ABB RAPID module: Mod1.mod

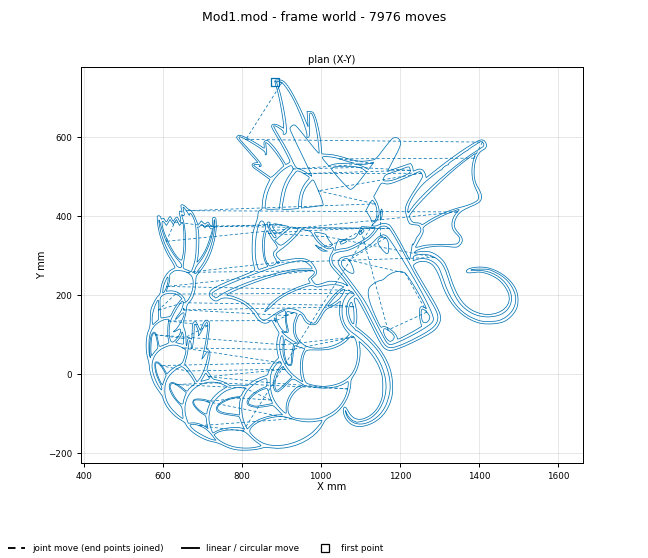
[picture p0: tool path of Mod1.mod in frame world, 7976 of 7976 moves have a stored position in this frame; points joined in program order, loops and branches not executed]
MODULE Module1
    !***********************************************************
    !
    ! Module:  Module1
    !
    ! Description:
    !   <Insert description here>
    !
    ! Author: ufabc
    !
    ! Version: 1.0
    !
    !***********************************************************


    !***********************************************************
    !
    ! Procedure main
    !
    !   This is the entry point of your program
    !
    !***********************************************************
    PROC main()
        !Add your code here
        CONST robtarget p0:=[[557.96,-192.62,509.20],[0.00299687,-0.165444,-0.986215,-0.000502744],[-1,0,0,0],[9E+09,9E+09,9E+09,9E+09,9E+09,9E+09]];	MoveJ Offs(p0,326.0,933.6, 10), v100, z1, tool0;
	MoveL Offs(p0,326.4428000000001,930.3582, 0), v100, z5, tool0;
	MoveL Offs(p0,326.7616,928.9504000000001, 0), v100, z5, tool0;
	MoveL Offs(p0,327.15,927.425, 0), v100, z5, tool0;
	MoveL Offs(p0,327.59839999999997,925.8095999999999, 0), v100, z5, tool0;
	MoveL Offs(p0,328.0972,924.1317999999999, 0), v100, z5, tool0;
	MoveL Offs(p0,328.63680000000005,922.4192, 0), v100, z5, tool0;
	MoveL Offs(p0,329.2076,920.6994000000001, 0), v100, z5, tool0;
	MoveL Offs(p0,329.8,919.0, 0), v100, z5, tool0;
	MoveL Offs(p0,331.7136,912.9074, 0), v100, z5, tool0;
	MoveL Offs(p0,333.90080000000006,904.3872000000003, 0), v100, z5, tool0;
	MoveL Offs(p0,336.25120000000004,894.0357999999999, 0), v100, z5, tool0;
	MoveL Offs(p0,338.6544,882.4496000000001, 0), v100, z5, tool0;
	MoveL Offs(p0,341.0,870.225, 0), v100, z5, tool0;
	MoveL Offs(p0,343.1776,857.9583999999999, 0), v100, z5, tool0;
	MoveL Offs(p0,345.0768,846.2461999999999, 0), v100, z5, tool0;
	MoveL Offs(p0,346.58720000000005,835.6848000000002, 0), v100, z5, tool0;
	MoveL Offs(p0,347.5984,826.8706, 0), v100, z5, tool0;
	MoveL Offs(p0,348.0,820.4, 0), v100, z5, tool0;
	MoveL Offs(p0,348.0,815.6, 0), v100, z5, tool0;
	MoveL Offs(p0,338.8,820.8, 0), v100, z5, tool0;
	MoveL Offs(p0,335.7876,822.3897999999999, 0), v100, z5, tool0;
	MoveL Offs(p0,332.98880000000014,823.6784000000001, 0), v100, z5, tool0;
	MoveL Offs(p0,330.40119999999996,824.6646000000001, 0), v100, z5, tool0;
	MoveL Offs(p0,328.0224,825.3471999999999, 0), v100, z5, tool0;
	MoveL Offs(p0,325.85,825.725, 0), v100, z5, tool0;
	MoveL Offs(p0,323.8816,825.7967999999998, 0), v100, z5, tool0;
	MoveL Offs(p0,322.11479999999995,825.5613999999999, 0), v100, z5, tool0;
	MoveL Offs(p0,320.54720000000003,825.0176000000001, 0), v100, z5, tool0;
	MoveL Offs(p0,319.1764,824.1641999999999, 0), v100, z5, tool0;
	MoveL Offs(p0,318.0,823.0, 0), v100, z5, tool0;
	MoveL Offs(p0,317.45279999999997,820.0318000000001, 0), v100, z5, tool0;
	MoveL Offs(p0,317.8976,818.4336000000001, 0), v100, z5, tool0;
	MoveL Offs(p0,318.7,816.425, 0), v100, z5, tool0;
	MoveL Offs(p0,319.8864,813.9424, 0), v100, z5, tool0;
	MoveL Offs(p0,321.4832,810.9222, 0), v100, z5, tool0;
	MoveL Offs(p0,323.51680000000005,807.3008000000001, 0), v100, z5, tool0;
	MoveL Offs(p0,326.01360000000005,803.0146000000001, 0), v100, z5, tool0;
	MoveL Offs(p0,329.0,798.0, 0), v100, z5, tool0;
	MoveL Offs(p0,333.77080000000007,789.9198000000001, 0), v100, z5, tool0;
	MoveL Offs(p0,338.63040000000007,781.4544000000002, 0), v100, z5, tool0;
	MoveL Offs(p0,343.43960000000004,772.8666000000001, 0), v100, z5, tool0;
	MoveL Offs(p0,348.05920000000003,764.4192, 0), v100, z5, tool0;
	MoveL Offs(p0,352.35,756.375, 0), v100, z5, tool0;
	MoveL Offs(p0,356.17279999999994,748.9967999999999, 0), v100, z5, tool0;
	MoveL Offs(p0,359.3884,742.5474, 0), v100, z5, tool0;
	MoveL Offs(p0,361.8576,737.2896000000001, 0), v100, z5, tool0;
	MoveL Offs(p0,363.44120000000004,733.4862, 0), v100, z5, tool0;
	MoveL Offs(p0,364.0,731.4, 0), v100, z5, tool0;
	MoveL Offs(p0,362.272,728.8313999999999, 0), v100, z5, tool0;
	MoveL Offs(p0,361.12,727.8448000000001, 0), v100, z5, tool0;
	MoveL Offs(p0,359.8,726.875, 0), v100, z5, tool0;
	MoveL Offs(p0,358.38399999999996,725.9712000000001, 0), v100, z5, tool0;
	MoveL Offs(p0,356.94399999999996,725.1826, 0), v100, z5, tool0;
	MoveL Offs(p0,355.552,724.5584000000001, 0), v100, z5, tool0;
	MoveL Offs(p0,354.28000000000003,724.1478000000001, 0), v100, z5, tool0;
	MoveL Offs(p0,353.2,724.0, 0), v100, z5, tool0;
	MoveL Offs(p0,351.7834,726.0466, 0), v100, z5, tool0;
	MoveL Offs(p0,350.82880000000006,727.5392000000002, 0), v100, z5, tool0;
	MoveL Offs(p0,349.675,729.375, 0), v100, z5, tool0;
	MoveL Offs(p0,348.34720000000004,731.5168, 0), v100, z5, tool0;
	MoveL Offs(p0,346.87059999999997,733.9273999999999, 0), v100, z5, tool0;
	MoveL Offs(p0,345.27040000000005,736.5696, 0), v100, z5, tool0;
	MoveL Offs(p0,343.5718,739.4062, 0), v100, z5, tool0;
	MoveL Offs(p0,341.8,742.4, 0), v100, z5, tool0;
	MoveL Offs(p0,339.87620000000004,745.5146000000001, 0), v100, z5, tool0;
	MoveL Offs(p0,337.73760000000004,748.8128000000003, 0), v100, z5, tool0;
	MoveL Offs(p0,335.4334,752.2262, 0), v100, z5, tool0;
	MoveL Offs(p0,333.0128,755.6864, 0), v100, z5, tool0;
	MoveL Offs(p0,330.525,759.125, 0), v100, z5, tool0;
	MoveL Offs(p0,328.0192,762.4735999999999, 0), v100, z5, tool0;
	MoveL Offs(p0,325.5446,765.6638, 0), v100, z5, tool0;
	MoveL Offs(p0,323.15040000000005,768.6272000000001, 0), v100, z5, tool0;
	MoveL Offs(p0,320.8858,771.2954000000001, 0), v100, z5, tool0;
	MoveL Offs(p0,318.8,773.6, 0), v100, z5, tool0;
	MoveL Offs(p0,315.7214,776.8180000000001, 0), v100, z5, tool0;
	MoveL Offs(p0,313.15520000000004,779.4240000000002, 0), v100, z5, tool0;
	MoveL Offs(p0,311.0258,781.466, 0), v100, z5, tool0;
	MoveL Offs(p0,309.2576,782.9920000000001, 0), v100, z5, tool0;
	MoveL Offs(p0,307.775,784.05, 0), v100, z5, tool0;
	MoveL Offs(p0,306.50239999999997,784.6879999999999, 0), v100, z5, tool0;
	MoveL Offs(p0,305.3642,784.954, 0), v100, z5, tool0;
	MoveL Offs(p0,304.2848,784.8960000000001, 0), v100, z5, tool0;
	MoveL Offs(p0,303.18860000000006,784.562, 0), v100, z5, tool0;
	MoveL Offs(p0,302.0,784.0, 0), v100, z5, tool0;
	MoveL Offs(p0,299.40079999999995,782.1351999999999, 0), v100, z5, tool0;
	MoveL Offs(p0,298.8736,781.3824000000001, 0), v100, z5, tool0;
	MoveL Offs(p0,298.5,780.5, 0), v100, z5, tool0;
	MoveL Offs(p0,298.27040000000005,779.4496, 0), v100, z5, tool0;
	MoveL Offs(p0,298.1752,778.1928, 0), v100, z5, tool0;
	MoveL Offs(p0,298.20480000000003,776.6912, 0), v100, z5, tool0;
	MoveL Offs(p0,298.3496,774.9064000000001, 0), v100, z5, tool0;
	MoveL Offs(p0,298.6,772.8, 0), v100, z5, tool0;
	MoveL Offs(p0,298.86120000000005,770.4126, 0), v100, z5, tool0;
	MoveL Offs(p0,299.0336000000001,768.5088000000003, 0), v100, z5, tool0;
	MoveL Offs(p0,299.1004,767.0562, 0), v100, z5, tool0;
	MoveL Offs(p0,299.0448,766.0224000000001, 0), v100, z5, tool0;
	MoveL Offs(p0,298.85,765.375, 0), v100, z5, tool0;
	MoveL Offs(p0,298.49920000000003,765.0815999999999, 0), v100, z5, tool0;
	MoveL Offs(p0,297.97560000000004,765.1098, 0), v100, z5, tool0;
	MoveL Offs(p0,297.2624,765.4272000000001, 0), v100, z5, tool0;
	MoveL Offs(p0,296.3428,766.0014, 0), v100, z5, tool0;
	MoveL Offs(p0,295.2,766.8, 0), v100, z5, tool0;
	MoveL Offs(p0,290.4552,770.0854000000002, 0), v100, z5, tool0;
	MoveL Offs(p0,285.0096000000001,773.6192000000003, 0), v100, z5, tool0;
	MoveL Offs(p0,279.0864,777.2778, 0), v100, z5, tool0;
	MoveL Offs(p0,272.90880000000004,780.9376000000001, 0), v100, z5, tool0;
	MoveL Offs(p0,266.7,784.475, 0), v100, z5, tool0;
	MoveL Offs(p0,260.6832,787.7663999999999, 0), v100, z5, tool0;
	MoveL Offs(p0,255.08159999999998,790.6881999999999, 0), v100, z5, tool0;
	MoveL Offs(p0,250.1184,793.1168, 0), v100, z5, tool0;
	MoveL Offs(p0,246.01680000000002,794.9286, 0), v100, z5, tool0;
	MoveL Offs(p0,243.0,796.0, 0), v100, z5, tool0;
	MoveL Offs(p0,240.78440000000006,796.5934000000001, 0), v100, z5, tool0;
	MoveL Offs(p0,238.90720000000005,797.0512000000001, 0), v100, z5, tool0;
	MoveL Offs(p0,237.3228,797.3697999999998, 0), v100, z5, tool0;
	MoveL Offs(p0,235.98559999999998,797.5456000000001, 0), v100, z5, tool0;
	MoveL Offs(p0,234.85,797.575, 0), v100, z5, tool0;
	MoveL Offs(p0,233.87039999999996,797.4544, 0), v100, z5, tool0;
	MoveL Offs(p0,233.0012,797.1802, 0), v100, z5, tool0;
	MoveL Offs(p0,232.1968,796.7488000000001, 0), v100, z5, tool0;
	MoveL Offs(p0,231.4116,796.1566, 0), v100, z5, tool0;
	MoveL Offs(p0,230.6,795.4, 0), v100, z5, tool0;
	MoveL Offs(p0,228.81260000000003,792.5002, 0), v100, z5, tool0;
	MoveL Offs(p0,229.43519999999998,790.8944, 0), v100, z5, tool0;
	MoveL Offs(p0,231.025,788.475, 0), v100, z5, tool0;
	MoveL Offs(p0,233.79680000000002,784.9456, 0), v100, z5, tool0;
	MoveL Offs(p0,237.9654,780.0098, 0), v100, z5, tool0;
	MoveL Offs(p0,243.74560000000002,773.3712000000002, 0), v100, z5, tool0;
	MoveL Offs(p0,251.35219999999998,764.7334000000001, 0), v100, z5, tool0;
	MoveL Offs(p0,261.0,753.8, 0), v100, z5, tool0;
	MoveL Offs(p0,282.8,729.0, 0), v100, z5, tool0;
	MoveL Offs(p0,276.0,728.0, 0), v100, z5, tool0;
	MoveL Offs(p0,273.33080000000007,727.4296, 0), v100, z5, tool0;
	MoveL Offs(p0,271.2064000000001,726.5808000000002, 0), v100, z5, tool0;
	MoveL Offs(p0,269.63160000000005,725.4871999999999, 0), v100, z5, tool0;
	MoveL Offs(p0,268.6112,724.1824, 0), v100, z5, tool0;
	MoveL Offs(p0,268.15,722.7, 0), v100, z5, tool0;
	MoveL Offs(p0,268.2528,721.0735999999999, 0), v100, z5, tool0;
	MoveL Offs(p0,268.9244,719.3368, 0), v100, z5, tool0;
	MoveL Offs(p0,270.1696,717.5232000000001, 0), v100, z5, tool0;
	MoveL Offs(p0,271.9932,715.6664000000001, 0), v100, z5, tool0;
	MoveL Offs(p0,274.4,713.8, 0), v100, z5, tool0;
	MoveL Offs(p0,277.2880000000001,711.8080000000002, 0), v100, z5, tool0;
	MoveL Offs(p0,279.206,710.452, 0), v100, z5, tool0;
	MoveL Offs(p0,281.37600000000003,708.9040000000001, 0), v100, z5, tool0;
	MoveL Offs(p0,283.75,707.2, 0), v100, z5, tool0;
	MoveL Offs(p0,286.28000000000003,705.376, 0), v100, z5, tool0;
	MoveL Offs(p0,288.918,703.4680000000001, 0), v100, z5, tool0;
	MoveL Offs(p0,291.61600000000004,701.5120000000001, 0), v100, z5, tool0;
	MoveL Offs(p0,294.326,699.5440000000001, 0), v100, z5, tool0;
	MoveL Offs(p0,297.0,697.6, 0), v100, z5, tool0;
	MoveL Offs(p0,313.2,685.8, 0), v100, z5, tool0;
	MoveL Offs(p0,306.6,672.4, 0), v100, z5, tool0;
	MoveL Offs(p0,304.44900000000007,667.78, 0), v100, z5, tool0;
	MoveL Offs(p0,302.4480000000001,662.8480000000002, 0), v100, z5, tool0;
	MoveL Offs(p0,300.61499999999995,657.676, 0), v100, z5, tool0;
	MoveL Offs(p0,298.96799999999996,652.336, 0), v100, z5, tool0;
	MoveL Offs(p0,297.525,646.9, 0), v100, z5, tool0;
	MoveL Offs(p0,296.304,641.44, 0), v100, z5, tool0;
	MoveL Offs(p0,295.323,636.028, 0), v100, z5, tool0;
	MoveL Offs(p0,294.6,630.7360000000001, 0), v100, z5, tool0;
	MoveL Offs(p0,294.15299999999996,625.6360000000001, 0), v100, z5, tool0;
	MoveL Offs(p0,294.0,620.8, 0), v100, z5, tool0;
	MoveL Offs(p0,293.9788,618.3684000000001, 0), v100, z5, tool0;
	MoveL Offs(p0,293.90240000000006,616.3232, 0), v100, z5, tool0;
	MoveL Offs(p0,293.7516,614.6188, 0), v100, z5, tool0;
	MoveL Offs(p0,293.5072,613.2096, 0), v100, z5, tool0;
	MoveL Offs(p0,293.15,612.05, 0), v100, z5, tool0;
	MoveL Offs(p0,292.6608,611.0944, 0), v100, z5, tool0;
	MoveL Offs(p0,292.0204,610.2972, 0), v100, z5, tool0;
	MoveL Offs(p0,291.2096,609.6128000000001, 0), v100, z5, tool0;
	MoveL Offs(p0,290.2092,608.9956, 0), v100, z5, tool0;
	MoveL Offs(p0,289.0,608.4, 0), v100, z5, tool0;
	MoveL Offs(p0,286.642,607.0985999999999, 0), v100, z5, tool0;
	MoveL Offs(p0,285.96000000000004,606.5952, 0), v100, z5, tool0;
	MoveL Offs(p0,285.35,606.075, 0), v100, z5, tool0;
	MoveL Offs(p0,284.824,605.5488, 0), v100, z5, tool0;
	MoveL Offs(p0,284.394,605.0274, 0), v100, z5, tool0;
	MoveL Offs(p0,284.072,604.5216, 0), v100, z5, tool0;
	MoveL Offs(p0,283.87,604.0422000000001, 0), v100, z5, tool0;
	MoveL Offs(p0,283.8,603.6, 0), v100, z5, tool0;
	MoveL Offs(p0,283.4896,600.7104, 0), v100, z5, tool0;
	MoveL Offs(p0,283.4,599.7, 0), v100, z5, tool0;
	MoveL Offs(p0,283.31039999999996,598.6176, 0), v100, z5, tool0;
	MoveL Offs(p0,283.2232,597.4848, 0), v100, z5, tool0;
	MoveL Offs(p0,283.1408,596.3232, 0), v100, z5, tool0;
	MoveL Offs(p0,283.0656,595.1544, 0), v100, z5, tool0;
	MoveL Offs(p0,283.0,594.0, 0), v100, z5, tool0;
	MoveL Offs(p0,282.44320000000005,590.9008000000001, 0), v100, z5, tool0;
	MoveL Offs(p0,281.9488,588.8142, 0), v100, z5, tool0;
	MoveL Offs(p0,281.3296,586.4384, 0), v100, z5, tool0;
	MoveL Offs(p0,280.6,583.825, 0), v100, z5, tool0;
	MoveL Offs(p0,279.77439999999996,581.0255999999999, 0), v100, z5, tool0;
	MoveL Offs(p0,278.8672,578.0917999999999, 0), v100, z5, tool0;
	MoveL Offs(p0,277.89279999999997,575.0752, 0), v100, z5, tool0;
	MoveL Offs(p0,276.8656,572.0274, 0), v100, z5, tool0;
	MoveL Offs(p0,275.8,569.0, 0), v100, z5, tool0;
	MoveL Offs(p0,274.1564000000001,564.3728000000001, 0), v100, z5, tool0;
	MoveL Offs(p0,272.8032000000001,560.3024000000001, 0), v100, z5, tool0;
	MoveL Offs(p0,271.7068,556.5655999999999, 0), v100, z5, tool0;
	MoveL Offs(p0,270.83360000000005,552.9392, 0), v100, z5, tool0;
	MoveL Offs(p0,270.15,549.2, 0), v100, z5, tool0;
	MoveL Offs(p0,269.62239999999997,545.1247999999999, 0), v100, z5, tool0;
	MoveL Offs(p0,269.2172,540.4904, 0), v100, z5, tool0;
	MoveL Offs(p0,268.9008,535.0735999999999, 0), v100, z5, tool0;
	MoveL Offs(p0,268.63960000000003,528.6512, 0), v100, z5, tool0;
	MoveL Offs(p0,268.4,521.0, 0), v100, z5, tool0;
	MoveL Offs(p0,268.2338000000001,512.9028000000001, 0), v100, z5, tool0;
	MoveL Offs(p0,268.22240000000005,505.56640000000016, 0), v100, z5, tool0;
	MoveL Offs(p0,268.37659999999994,498.8636, 0), v100, z5, tool0;
	MoveL Offs(p0,268.7072,492.66720000000004, 0), v100, z5, tool0;
	MoveL Offs(p0,269.225,486.85, 0), v100, z5, tool0;
	MoveL Offs(p0,269.94079999999997,481.2848, 0), v100, z5, tool0;
	MoveL Offs(p0,270.8654,475.84439999999995, 0), v100, z5, tool0;
	MoveL Offs(p0,272.00960000000003,470.4016, 0), v100, z5, tool0;
	MoveL Offs(p0,273.3842,464.8292, 0), v100, z5, tool0;
	MoveL Offs(p0,275.0,459.0, 0), v100, z5, tool0;
	MoveL Offs(p0,275.0176,456.8880000000001, 0), v100, z5, tool0;
	MoveL Offs(p0,274.30339999999995,455.85, 0), v100, z5, tool0;
	MoveL Offs(p0,272.93280000000004,454.72799999999995, 0), v100, z5, tool0;
	MoveL Offs(p0,270.775,453.45, 0), v100, z5, tool0;
	MoveL Offs(p0,267.6992,451.9440000000001, 0), v100, z5, tool0;
	MoveL Offs(p0,263.57460000000003,450.13800000000003, 0), v100, z5, tool0;
	MoveL Offs(p0,258.2704,447.96000000000004, 0), v100, z5, tool0;
	MoveL Offs(p0,251.6558,445.338, 0), v100, z5, tool0;
	MoveL Offs(p0,243.6,442.2, 0), v100, z5, tool0;
	MoveL Offs(p0,230.11380000000003,436.89400000000006, 0), v100, z5, tool0;
	MoveL Offs(p0,217.95840000000004,432.00800000000015, 0), v100, z5, tool0;
	MoveL Offs(p0,207.10859999999997,427.53000000000003, 0), v100, z5, tool0;
	MoveL Offs(p0,197.5392,423.44800000000004, 0), v100, z5, tool0;
	MoveL Offs(p0,189.225,419.75, 0), v100, z5, tool0;
	MoveL Offs(p0,182.14079999999998,416.424, 0), v100, z5, tool0;
	MoveL Offs(p0,176.2614,413.45799999999997, 0), v100, z5, tool0;
	MoveL Offs(p0,171.5616,410.84, 0), v100, z5, tool0;
	MoveL Offs(p0,168.0162,408.558, 0), v100, z5, tool0;
	MoveL Offs(p0,165.6,406.6, 0), v100, z5, tool0;
	MoveL Offs(p0,163.50000000000003,404.2816000000001, 0), v100, z5, tool0;
	MoveL Offs(p0,161.88000000000005,401.9008000000001, 0), v100, z5, tool0;
	MoveL Offs(p0,160.74,399.47919999999993, 0), v100, z5, tool0;
	MoveL Offs(p0,160.08,397.0384, 0), v100, z5, tool0;
	MoveL Offs(p0,159.9,394.6, 0), v100, z5, tool0;
	MoveL Offs(p0,160.2,392.18559999999997, 0), v100, z5, tool0;
	MoveL Offs(p0,160.98000000000002,389.81679999999994, 0), v100, z5, tool0;
	MoveL Offs(p0,162.24,387.5152, 0), v100, z5, tool0;
	MoveL Offs(p0,163.98000000000002,385.30240000000003, 0), v100, z5, tool0;
	MoveL Offs(p0,166.2,383.2, 0), v100, z5, tool0;
	MoveL Offs(p0,168.3522,381.51400000000007, 0), v100, z5, tool0;
	MoveL Offs(p0,170.38560000000007,380.17600000000004, 0), v100, z5, tool0;
	MoveL Offs(p0,172.3254,379.18600000000004, 0), v100, z5, tool0;
	MoveL Offs(p0,174.1968,378.544, 0), v100, z5, tool0;
	MoveL Offs(p0,176.025,378.25, 0), v100, z5, tool0;
	MoveL Offs(p0,177.83520000000001,378.304, 0), v100, z5, tool0;
	MoveL Offs(p0,179.65259999999998,378.706, 0), v100, z5, tool0;
	MoveL Offs(p0,181.50240000000002,379.456, 0), v100, z5, tool0;
	MoveL Offs(p0,183.40980000000002,380.554, 0), v100, z5, tool0;
	MoveL Offs(p0,185.4,382.0, 0), v100, z5, tool0;
	MoveL Offs(p0,189.10640000000004,384.06820000000005, 0), v100, z5, tool0;
	MoveL Offs(p0,193.76320000000004,385.36960000000005, 0), v100, z5, tool0;
	MoveL Offs(p0,199.21679999999998,385.9294, 0), v100, z5, tool0;
	MoveL Offs(p0,205.31360000000004,385.7728000000001, 0), v100, z5, tool0;
	MoveL Offs(p0,211.9,384.925, 0), v100, z5, tool0;
	MoveL Offs(p0,218.82240000000002,383.4112, 0), v100, z5, tool0;
	MoveL Offs(p0,225.9272,381.2566, 0), v100, z5, tool0;
	MoveL Offs(p0,233.06080000000003,378.48640000000006, 0), v100, z5, tool0;
	MoveL Offs(p0,240.06959999999998,375.12579999999997, 0), v100, z5, tool0;
	MoveL Offs(p0,246.8,371.2, 0), v100, z5, tool0;
	MoveL Offs(p0,250.31440000000003,368.80140000000006, 0), v100, z5, tool0;
	MoveL Offs(p0,253.77120000000005,366.1712000000001, 0), v100, z5, tool0;
	MoveL Offs(p0,257.1608,363.31780000000003, 0), v100, z5, tool0;
	MoveL Offs(p0,260.47360000000003,360.2496, 0), v100, z5, tool0;
	MoveL Offs(p0,263.7,356.975, 0), v100, z5, tool0;
	MoveL Offs(p0,266.8304,353.50239999999997, 0), v100, z5, tool0;
	MoveL Offs(p0,269.85519999999997,349.8402, 0), v100, z5, tool0;
	MoveL Offs(p0,272.76480000000004,345.9968, 0), v100, z5, tool0;
	MoveL Offs(p0,275.5496,341.98060000000004, 0), v100, z5, tool0;
	MoveL Offs(p0,278.2,337.8, 0), v100, z5, tool0;
	MoveL Offs(p0,281.2044,333.5006000000001, 0), v100, z5, tool0;
	MoveL Offs(p0,284.4272,329.85280000000006, 0), v100, z5, tool0;
	MoveL Offs(p0,287.82280000000003,326.8722, 0), v100, z5, tool0;
	MoveL Offs(p0,291.3456,324.5744, 0), v100, z5, tool0;
	MoveL Offs(p0,294.95,322.975, 0), v100, z5, tool0;
	MoveL Offs(p0,298.5904,322.08959999999996, 0), v100, z5, tool0;
	MoveL Offs(p0,302.2212,321.93379999999996, 0), v100, z5, tool0;
	MoveL Offs(p0,305.7968,322.5232, 0), v100, z5, tool0;
	MoveL Offs(p0,309.27160000000003,323.87340000000006, 0), v100, z5, tool0;
	MoveL Offs(p0,312.6,326.0, 0), v100, z5, tool0;
	MoveL Offs(p0,317.8,330.2, 0), v100, z5, tool0;
	MoveL Offs(p0,322.8,320.6, 0), v100, z5, tool0;
	MoveL Offs(p0,324.64480000000015,317.2416000000002, 0), v100, z5, tool0;
	MoveL Offs(p0,325.6601999999999,315.4394, 0), v100, z5, tool0;
	MoveL Offs(p0,326.71040000000005,313.6048, 0), v100, z5, tool0;
	MoveL Offs(p0,327.775,311.775, 0), v100, z5, tool0;
	MoveL Offs(p0,328.83360000000005,309.9872, 0), v100, z5, tool0;
	MoveL Offs(p0,329.8658,308.2786, 0), v100, z5, tool0;
	MoveL Offs(p0,330.85120000000006,306.68640000000005, 0), v100, z5, tool0;
	MoveL Offs(p0,331.7694,305.2478, 0), v100, z5, tool0;
	MoveL Offs(p0,332.6,304.0, 0), v100, z5, tool0;
	MoveL Offs(p0,334.74720000000013,300.7248000000001, 0), v100, z5, tool0;
	MoveL Offs(p0,335.4638,299.4172, 0), v100, z5, tool0;
	MoveL Offs(p0,335.95360000000005,298.2464, 0), v100, z5, tool0;
	MoveL Offs(p0,336.225,297.15, 0), v100, z5, tool0;
	MoveL Offs(p0,336.2864,296.0656, 0), v100, z5, tool0;
	MoveL Offs(p0,336.1462,294.9308, 0), v100, z5, tool0;
	MoveL Offs(p0,335.81280000000004,293.68320000000006, 0), v100, z5, tool0;
	MoveL Offs(p0,335.2946,292.2604, 0), v100, z5, tool0;
	MoveL Offs(p0,334.6,290.6, 0), v100, z5, tool0;
	MoveL Offs(p0,333.38820000000004,287.2198, 0), v100, z5, tool0;
	MoveL Offs(p0,332.3936000000001,283.4784000000001, 0), v100, z5, tool0;
	MoveL Offs(p0,331.6174,279.4346, 0), v100, z5, tool0;
	MoveL Offs(p0,331.0608,275.1472, 0), v100, z5, tool0;
	MoveL Offs(p0,330.725,270.675, 0), v100, z5, tool0;
	MoveL Offs(p0,330.6112,266.0768, 0), v100, z5, tool0;
	MoveL Offs(p0,330.7206,261.4114, 0), v100, z5, tool0;
	MoveL Offs(p0,331.0544,256.73760000000004, 0), v100, z5, tool0;
	MoveL Offs(p0,331.6138,252.11419999999998, 0), v100, z5, tool0;
	MoveL Offs(p0,332.4,247.6, 0), v100, z5, tool0;
	MoveL Offs(p0,335.2,234.2, 0), v100, z5, tool0;
	MoveL Offs(p0,327.6,226.6, 0), v100, z5, tool0;
	MoveL Offs(p0,325.253,224.04980000000006, 0), v100, z5, tool0;
	MoveL Offs(p0,322.72000000000014,220.83840000000004, 0), v100, z5, tool0;
	MoveL Offs(p0,320.10299999999995,217.1446, 0), v100, z5, tool0;
	MoveL Offs(p0,317.504,213.14720000000003, 0), v100, z5, tool0;
	MoveL Offs(p0,315.025,209.025, 0), v100, z5, tool0;
	MoveL Offs(p0,312.768,204.95680000000002, 0), v100, z5, tool0;
	MoveL Offs(p0,310.83500000000004,201.1214, 0), v100, z5, tool0;
	MoveL Offs(p0,309.32800000000003,197.69760000000002, 0), v100, z5, tool0;
	MoveL Offs(p0,308.349,194.8642, 0), v100, z5, tool0;
	MoveL Offs(p0,308.0,192.8, 0), v100, z5, tool0;
	MoveL Offs(p0,305.55,190.325, 0), v100, z5, tool0;
	MoveL Offs(p0,304.5872,189.8048, 0), v100, z5, tool0;
	MoveL Offs(p0,303.5116,189.3014, 0), v100, z5, tool0;
	MoveL Offs(p0,302.3424,188.8256, 0), v100, z5, tool0;
	MoveL Offs(p0,301.09880000000004,188.3882, 0), v100, z5, tool0;
	MoveL Offs(p0,299.8,188.0, 0), v100, z5, tool0;
	MoveL Offs(p0,295.9290000000001,186.8418, 0), v100, z5, tool0;
	MoveL Offs(p0,291.92,185.43040000000005, 0), v100, z5, tool0;
	MoveL Offs(p0,287.83900000000006,183.8006, 0), v100, z5, tool0;
	MoveL Offs(p0,283.752,181.98720000000003, 0), v100, z5, tool0;
	MoveL Offs(p0,279.725,180.025, 0), v100, z5, tool0;
	MoveL Offs(p0,275.82399999999996,177.9488, 0), v100, z5, tool0;
	MoveL Offs(p0,272.11499999999995,175.79339999999996, 0), v100, z5, tool0;
	MoveL Offs(p0,268.66400000000004,173.5936, 0), v100, z5, tool0;
	MoveL Offs(p0,265.53700000000003,171.38420000000002, 0), v100, z5, tool0;
	MoveL Offs(p0,262.8,169.2, 0), v100, z5, tool0;
	MoveL Offs(p0,259.1408000000001,166.16800000000003, 0), v100, z5, tool0;
	MoveL Offs(p0,257.65919999999994,165.132, 0), v100, z5, tool0;
	MoveL Offs(p0,256.27840000000003,164.38400000000001, 0), v100, z5, tool0;
	MoveL Offs(p0,254.9,163.9, 0), v100, z5, tool0;
	MoveL Offs(p0,253.42559999999997,163.656, 0), v100, z5, tool0;
	MoveL Offs(p0,251.75679999999997,163.628, 0), v100, z5, tool0;
	MoveL Offs(p0,249.79520000000002,163.792, 0), v100, z5, tool0;
	MoveL Offs(p0,247.4424,164.12400000000002, 0), v100, z5, tool0;
	MoveL Offs(p0,244.6,164.6, 0), v100, z5, tool0;
	MoveL Offs(p0,240.55040000000014,165.08000000000004, 0), v100, z5, tool0;
	MoveL Offs(p0,238.40259999999998,165.22999999999996, 0), v100, z5, tool0;
	MoveL Offs(p0,236.2032,165.32, 0), v100, z5, tool0;
	MoveL Offs(p0,233.975,165.35, 0), v100, z5, tool0;
	MoveL Offs(p0,231.74079999999998,165.32, 0), v100, z5, tool0;
	MoveL Offs(p0,229.52339999999998,165.22999999999996, 0), v100, z5, tool0;
	MoveL Offs(p0,227.34560000000002,165.08, 0), v100, z5, tool0;
	MoveL Offs(p0,225.23020000000002,164.87000000000003, 0), v100, z5, tool0;
	MoveL Offs(p0,223.2,164.6, 0), v100, z5, tool0;
	MoveL Offs(p0,220.54840000000007,164.12760000000003, 0), v100, z5, tool0;
	MoveL Offs(p0,218.30720000000005,163.79680000000005, 0), v100, z5, tool0;
	MoveL Offs(p0,216.40680000000003,163.6172, 0), v100, z5, tool0;
	MoveL Offs(p0,214.77759999999998,163.5984, 0), v100, z5, tool0;
	MoveL Offs(p0,213.35,163.75, 0), v100, z5, tool0;
	MoveL Offs(p0,212.0544,164.08160000000004, 0), v100, z5, tool0;
	MoveL Offs(p0,210.8212,164.60279999999997, 0), v100, z5, tool0;
	MoveL Offs(p0,209.5808,165.32319999999999, 0), v100, z5, tool0;
	MoveL Offs(p0,208.2636,166.25240000000002, 0), v100, z5, tool0;
	MoveL Offs(p0,206.8,167.4, 0), v100, z5, tool0;
	MoveL Offs(p0,202.48000000000005,170.23680000000004, 0), v100, z5, tool0;
	MoveL Offs(p0,199.834,171.6012, 0), v100, z5, tool0;
	MoveL Offs(p0,196.912,172.9104, 0), v100, z5, tool0;
	MoveL Offs(p0,193.75,174.15, 0), v100, z5, tool0;
	MoveL Offs(p0,190.38400000000001,175.3056, 0), v100, z5, tool0;
	MoveL Offs(p0,186.85,176.3628, 0), v100, z5, tool0;
	MoveL Offs(p0,183.18400000000003,177.30720000000002, 0), v100, z5, tool0;
	MoveL Offs(p0,179.42200000000003,178.1244, 0), v100, z5, tool0;
	MoveL Offs(p0,175.6,178.8, 0), v100, z5, tool0;
	MoveL Offs(p0,172.40960000000004,179.55200000000005, 0), v100, z5, tool0;
	MoveL Offs(p0,171.0694,180.078, 0), v100, z5, tool0;
	MoveL Offs(p0,169.85280000000003,180.73600000000002, 0), v100, z5, tool0;
	MoveL Offs(p0,168.725,181.55, 0), v100, z5, tool0;
	MoveL Offs(p0,167.6512,182.54399999999998, 0), v100, z5, tool0;
	MoveL Offs(p0,166.5966,183.74200000000002, 0), v100, z5, tool0;
	MoveL Offs(p0,165.52640000000002,185.168, 0), v100, z5, tool0;
	MoveL Offs(p0,164.4058,186.846, 0), v100, z5, tool0;
	MoveL Offs(p0,163.2,188.8, 0), v100, z5, tool0;
	MoveL Offs(p0,161.46720000000005,191.57440000000003, 0), v100, z5, tool0;
	MoveL Offs(p0,160.5828,192.9346, 0), v100, z5, tool0;
	MoveL Offs(p0,159.7056,194.24320000000003, 0), v100, z5, tool0;
	MoveL Offs(p0,158.85,195.475, 0), v100, z5, tool0;
	MoveL Offs(p0,158.03040000000001,196.6048, 0), v100, z5, tool0;
	MoveL Offs(p0,157.2612,197.60739999999998, 0), v100, z5, tool0;
	MoveL Offs(p0,156.5568,198.4576, 0), v100, z5, tool0;
	MoveL Offs(p0,155.93160000000003,199.1302, 0), v100, z5, tool0;
	MoveL Offs(p0,155.4,199.6, 0), v100, z5, tool0;
	MoveL Offs(p0,154.0176,201.89679999999998, 0), v100, z5, tool0;
	MoveL Offs(p0,153.91520000000003,203.04960000000003, 0), v100, z5, tool0;
	MoveL Offs(p0,154.0,204.5, 0), v100, z5, tool0;
	MoveL Offs(p0,154.27679999999998,206.3104, 0), v100, z5, tool0;
	MoveL Offs(p0,154.75039999999998,208.54319999999998, 0), v100, z5, tool0;
	MoveL Offs(p0,155.4256,211.26080000000002, 0), v100, z5, tool0;
	MoveL Offs(p0,156.30720000000002,214.52560000000003, 0), v100, z5, tool0;
	MoveL Offs(p0,157.4,218.4, 0), v100, z5, tool0;
	MoveL Offs(p0,158.9116,224.1442, 0), v100, z5, tool0;
	MoveL Offs(p0,160.08480000000003,229.48160000000007, 0), v100, z5, tool0;
	MoveL Offs(p0,160.91720000000004,234.38939999999997, 0), v100, z5, tool0;
	MoveL Offs(p0,161.40640000000002,238.84480000000002, 0), v100, z5, tool0;
	MoveL Offs(p0,161.55,242.825, 0), v100, z5, tool0;
	MoveL Offs(p0,161.3456,246.30720000000002, 0), v100, z5, tool0;
	MoveL Offs(p0,160.7908,249.26859999999996, 0), v100, z5, tool0;
	MoveL Offs(p0,159.8832,251.68640000000005, 0), v100, z5, tool0;
	MoveL Offs(p0,158.62040000000002,253.5378, 0), v100, z5, tool0;
	MoveL Offs(p0,157.0,254.8, 0), v100, z5, tool0;
	MoveL Offs(p0,154.5584,256.0928, 0), v100, z5, tool0;
	MoveL Offs(p0,154.05,256.35, 0), v100, z5, tool0;
	MoveL Offs(p0,153.60160000000002,256.5712, 0), v100, z5, tool0;
	MoveL Offs(p0,153.2228,256.7516, 0), v100, z5, tool0;
	MoveL Offs(p0,152.92320000000004,256.88640000000004, 0), v100, z5, tool0;
	MoveL Offs(p0,152.71240000000003,256.9708, 0), v100, z5, tool0;
	MoveL Offs(p0,152.6,257.0, 0), v100, z5, tool0;
	MoveL Offs(p0,152.95,259.975, 0), v100, z5, tool0;
	MoveL Offs(p0,153.14719999999997,261.1472, 0), v100, z5, tool0;
	MoveL Offs(p0,153.3756,262.45860000000005, 0), v100, z5, tool0;
	MoveL Offs(p0,153.6304,263.88640000000004, 0), v100, z5, tool0;
	MoveL Offs(p0,153.90680000000003,265.4078, 0), v100, z5, tool0;
	MoveL Offs(p0,154.2,267.0, 0), v100, z5, tool0;
	MoveL Offs(p0,155.00640000000004,271.37280000000004, 0), v100, z5, tool0;
	MoveL Offs(p0,155.46359999999999,274.21619999999996, 0), v100, z5, tool0;
	MoveL Offs(p0,155.9472,277.40639999999996, 0), v100, z5, tool0;
	MoveL Offs(p0,156.45,280.875, 0), v100, z5, tool0;
	MoveL Offs(p0,156.96479999999997,284.5536, 0), v100, z5, tool0;
	MoveL Offs(p0,157.4844,288.3738, 0), v100, z5, tool0;
	MoveL Offs(p0,158.0016,292.26720000000006, 0), v100, z5, tool0;
	MoveL Offs(p0,158.50920000000002,296.16540000000003, 0), v100, z5, tool0;
	MoveL Offs(p0,159.0,300.0, 0), v100, z5, tool0;
	MoveL Offs(p0,159.6474,305.7074000000001, 0), v100, z5, tool0;
	MoveL Offs(p0,160.14720000000003,310.4272000000001, 0), v100, z5, tool0;
	MoveL Offs(p0,160.49579999999997,314.2758, 0), v100, z5, tool0;
	MoveL Offs(p0,160.6896,317.36960000000005, 0), v100, z5, tool0;
	MoveL Offs(p0,160.725,319.825, 0), v100, z5, tool0;
	MoveL Offs(p0,160.59840000000003,321.7584, 0), v100, z5, tool0;
	MoveL Offs(p0,160.3062,323.2862, 0), v100, z5, tool0;
	MoveL Offs(p0,159.84480000000002,324.5248, 0), v100, z5, tool0;
	MoveL Offs(p0,159.2106,325.5906, 0), v100, z5, tool0;
	MoveL Offs(p0,158.4,326.6, 0), v100, z5, tool0;
	MoveL Offs(p0,155.0448,329.3008000000001, 0), v100, z5, tool0;
	MoveL Offs(p0,153.43919999999997,329.7842, 0), v100, z5, tool0;
	MoveL Offs(p0,151.8624,329.6784, 0), v100, z5, tool0;
	MoveL Offs(p0,150.3,328.975, 0), v100, z5, tool0;
	MoveL Offs(p0,148.7376,327.6656, 0), v100, z5, tool0;
	MoveL Offs(p0,147.1608,325.7418, 0), v100, z5, tool0;
	MoveL Offs(p0,145.5552,323.1952, 0), v100, z5, tool0;
	MoveL Offs(p0,143.90640000000002,320.0174, 0), v100, z5, tool0;
	MoveL Offs(p0,142.2,316.2, 0), v100, z5, tool0;
	MoveL Offs(p0,137.0,303.4, 0), v100, z5, tool0;
	MoveL Offs(p0,132.0,314.6, 0), v100, z5, tool0;
	MoveL Offs(p0,130.38880000000003,318.16640000000007, 0), v100, z5, tool0;
	MoveL Offs(p0,129.5682,319.7966, 0), v100, z5, tool0;
	MoveL Offs(p0,128.7584,321.2912, 0), v100, z5, tool0;
	MoveL Offs(p0,127.975,322.625, 0), v100, z5, tool0;
	MoveL Offs(p0,127.23359999999998,323.77279999999996, 0), v100, z5, tool0;
	MoveL Offs(p0,126.5498,324.7094, 0), v100, z5, tool0;
	MoveL Offs(p0,125.9392,325.4096, 0), v100, z5, tool0;
	MoveL Offs(p0,125.4174,325.8482, 0), v100, z5, tool0;
	MoveL Offs(p0,125.0,326.0, 0), v100, z5, tool0;
	MoveL Offs(p0,122.09280000000001,325.41280000000006, 0), v100, z5, tool0;
	MoveL Offs(p0,120.88520000000001,324.7562, 0), v100, z5, tool0;
	MoveL Offs(p0,119.83840000000001,323.8464, 0), v100, z5, tool0;
	MoveL Offs(p0,118.95,322.675, 0), v100, z5, tool0;
	MoveL Offs(p0,118.21759999999999,321.23359999999997, 0), v100, z5, tool0;
	MoveL Offs(p0,117.63879999999999,319.5138, 0), v100, z5, tool0;
	MoveL Offs(p0,117.2112,317.5072, 0), v100, z5, tool0;
	MoveL Offs(p0,116.9324,315.2054, 0), v100, z5, tool0;
	MoveL Offs(p0,116.8,312.6, 0), v100, z5, tool0;
	MoveL Offs(p0,116.7168,306.7532, 0), v100, z5, tool0;
	MoveL Offs(p0,116.59040000000002,301.36960000000005, 0), v100, z5, tool0;
	MoveL Offs(p0,116.42559999999999,296.5044, 0), v100, z5, tool0;
	MoveL Offs(p0,116.22720000000001,292.2128, 0), v100, z5, tool0;
	MoveL Offs(p0,116.0,288.55, 0), v100, z5, tool0;
	MoveL Offs(p0,115.7488,285.5712, 0), v100, z5, tool0;
	MoveL Offs(p0,115.47840000000001,283.33160000000004, 0), v100, z5, tool0;
	MoveL Offs(p0,115.19360000000002,281.88640000000004, 0), v100, z5, tool0;
	MoveL Offs(p0,114.8992,281.29080000000005, 0), v100, z5, tool0;
	MoveL Offs(p0,114.6,281.6, 0), v100, z5, tool0;
	MoveL Offs(p0,112.21679999999999,283.64480000000003, 0), v100, z5, tool0;
	MoveL Offs(p0,111.08960000000002,283.88160000000005, 0), v100, z5, tool0;
	MoveL Offs(p0,109.9,283.9, 0), v100, z5, tool0;
	MoveL Offs(p0,108.7104,283.7024, 0), v100, z5, tool0;
	MoveL Offs(p0,107.58319999999999,283.2912, 0), v100, z5, tool0;
	MoveL Offs(p0,106.5808,282.66880000000003, 0), v100, z5, tool0;
	MoveL Offs(p0,105.76559999999999,281.8376, 0), v100, z5, tool0;
	MoveL Offs(p0,105.2,280.8, 0), v100, z5, tool0;
	MoveL Offs(p0,104.6762,278.721, 0), v100, z5, tool0;
	MoveL Offs(p0,104.5184,277.872, 0), v100, z5, tool0;
	MoveL Offs(p0,104.375,276.975, 0), v100, z5, tool0;
	MoveL Offs(p0,104.24960000000002,276.04799999999994, 0), v100, z5, tool0;
	MoveL Offs(p0,104.14579999999998,275.10900000000004, 0), v100, z5, tool0;
	MoveL Offs(p0,104.0672,274.17600000000004, 0), v100, z5, tool0;
	MoveL Offs(p0,104.0174,273.267, 0), v100, z5, tool0;
	MoveL Offs(p0,104.0,272.4, 0), v100, z5, tool0;
	MoveL Offs(p0,103.80559999999998,269.65680000000003, 0), v100, z5, tool0;
	MoveL Offs(p0,103.66720000000001,268.7616, 0), v100, z5, tool0;
	MoveL Offs(p0,103.5,267.9, 0), v100, z5, tool0;
	MoveL Offs(p0,103.30879999999999,267.08639999999997, 0), v100, z5, tool0;
	MoveL Offs(p0,103.0984,266.3352, 0), v100, z5, tool0;
	MoveL Offs(p0,102.87360000000001,265.6608, 0), v100, z5, tool0;
	MoveL Offs(p0,102.6392,265.07759999999996, 0), v100, z5, tool0;
	MoveL Offs(p0,102.4,264.6, 0), v100, z5, tool0;
	MoveL Offs(p0,101.54880000000001,266.6544, 0), v100, z5, tool0;
	MoveL Offs(p0,101.375,268.125, 0), v100, z5, tool0;
	MoveL Offs(p0,101.2192,269.9136, 0), v100, z5, tool0;
	MoveL Offs(p0,101.0826,271.9878, 0), v100, z5, tool0;
	MoveL Offs(p0,100.96640000000001,274.3152, 0), v100, z5, tool0;
	MoveL Offs(p0,100.87180000000001,276.8634, 0), v100, z5, tool0;
	MoveL Offs(p0,100.8,279.6, 0), v100, z5, tool0;
	MoveL Offs(p0,100.76380000000002,283.04460000000006, 0), v100, z5, tool0;
	MoveL Offs(p0,100.65440000000002,286.3008000000001, 0), v100, z5, tool0;
	MoveL Offs(p0,100.4706,289.37219999999996, 0), v100, z5, tool0;
	MoveL Offs(p0,100.21120000000002,292.2624, 0), v100, z5, tool0;
	MoveL Offs(p0,99.875,294.975, 0), v100, z5, tool0;
	MoveL Offs(p0,99.46079999999999,297.5136, 0), v100, z5, tool0;
	MoveL Offs(p0,98.9674,299.8818, 0), v100, z5, tool0;
	MoveL Offs(p0,98.3936,302.08320000000003, 0), v100, z5, tool0;
	MoveL Offs(p0,97.7382,304.1214, 0), v100, z5, tool0;
	MoveL Offs(p0,97.0,306.0, 0), v100, z5, tool0;
	MoveL Offs(p0,95.81200000000001,309.19780000000003, 0), v100, z5, tool0;
	MoveL Offs(p0,94.88800000000002,312.11840000000007, 0), v100, z5, tool0;
	MoveL Offs(p0,94.228,314.83259999999996, 0), v100, z5, tool0;
	MoveL Offs(p0,93.83200000000001,317.41120000000006, 0), v100, z5, tool0;
	MoveL Offs(p0,93.7,319.925, 0), v100, z5, tool0;
	MoveL Offs(p0,93.83200000000001,322.44480000000004, 0), v100, z5, tool0;
	MoveL Offs(p0,94.228,325.0414, 0), v100, z5, tool0;
	MoveL Offs(p0,94.888,327.78560000000004, 0), v100, z5, tool0;
	MoveL Offs(p0,95.81200000000001,330.7482, 0), v100, z5, tool0;
	MoveL Offs(p0,97.0,334.0, 0), v100, z5, tool0;
	MoveL Offs(p0,98.11040000000001,337.4944000000001, 0), v100, z5, tool0;
	MoveL Offs(p0,98.6686,339.5476, 0), v100, z5, tool0;
	MoveL Offs(p0,99.2112,341.74719999999996, 0), v100, z5, tool0;
	MoveL Offs(p0,99.725,344.05, 0), v100, z5, tool0;
	MoveL Offs(p0,100.19680000000001,346.41279999999995, 0), v100, z5, tool0;
	MoveL Offs(p0,100.6134,348.7924, 0), v100, z5, tool0;
	MoveL Offs(p0,100.9616,351.1456, 0), v100, z5, tool0;
	MoveL Offs(p0,101.22820000000002,353.42920000000004, 0), v100, z5, tool0;
	MoveL Offs(p0,101.4,355.6, 0), v100, z5, tool0;
	MoveL Offs(p0,101.71020000000001,358.5570000000001, 0), v100, z5, tool0;
	MoveL Offs(p0,102.05760000000002,361.11200000000014, 0), v100, z5, tool0;
	MoveL Offs(p0,102.4674,363.33099999999996, 0), v100, z5, tool0;
	MoveL Offs(p0,102.96480000000001,365.28000000000003, 0), v100, z5, tool0;
	MoveL Offs(p0,103.575,367.025, 0), v100, z5, tool0;
	MoveL Offs(p0,104.3232,368.632, 0), v100, z5, tool0;
	MoveL Offs(p0,105.2346,370.16700000000003, 0), v100, z5, tool0;
	MoveL Offs(p0,106.3344,371.696, 0), v100, z5, tool0;
	MoveL Offs(p0,107.6478,373.285, 0), v100, z5, tool0;
	MoveL Offs(p0,109.2,375.0, 0), v100, z5, tool0;
	MoveL Offs(p0,112.06180000000002,378.39560000000006, 0), v100, z5, tool0;
	MoveL Offs(p0,114.64640000000004,382.10080000000005, 0), v100, z5, tool0;
	MoveL Offs(p0,116.9526,386.11319999999995, 0), v100, z5, tool0;
	MoveL Offs(p0,118.97920000000002,390.4304, 0), v100, z5, tool0;
	MoveL Offs(p0,120.725,395.05, 0), v100, z5, tool0;
	MoveL Offs(p0,122.18879999999999,399.9696, 0), v100, z5, tool0;
	MoveL Offs(p0,123.3694,405.18679999999995, 0), v100, z5, tool0;
	MoveL Offs(p0,124.26559999999999,410.6992, 0), v100, z5, tool0;
	MoveL Offs(p0,124.87620000000001,416.5044, 0), v100, z5, tool0;
	MoveL Offs(p0,125.2,422.6, 0), v100, z5, tool0;
	MoveL Offs(p0,125.33380000000002,426.57480000000004, 0), v100, z5, tool0;
	MoveL Offs(p0,125.50240000000004,430.01440000000014, 0), v100, z5, tool0;
	MoveL Offs(p0,125.7166,432.9716, 0), v100, z5, tool0;
	MoveL Offs(p0,125.9872,435.49920000000003, 0), v100, z5, tool0;
	MoveL Offs(p0,126.325,437.65, 0), v100, z5, tool0;
	MoveL Offs(p0,126.7408,439.4768, 0), v100, z5, tool0;
	MoveL Offs(p0,127.24539999999999,441.03239999999994, 0), v100, z5, tool0;
	MoveL Offs(p0,127.84960000000001,442.3696, 0), v100, z5, tool0;
	MoveL Offs(p0,128.5642,443.5412, 0), v100, z5, tool0;
	MoveL Offs(p0,129.4,444.6, 0), v100, z5, tool0;
	MoveL Offs(p0,132.42540000000002,448.14160000000004, 0), v100, z5, tool0;
	MoveL Offs(p0,135.57920000000004,452.10080000000005, 0), v100, z5, tool0;
	MoveL Offs(p0,138.7978,456.37919999999997, 0), v100, z5, tool0;
	MoveL Offs(p0,142.0176,460.87840000000006, 0), v100, z5, tool0;
	MoveL Offs(p0,145.175,465.5, 0), v100, z5, tool0;
	MoveL Offs(p0,148.2064,470.1456, 0), v100, z5, tool0;
	MoveL Offs(p0,151.0482,474.7168, 0), v100, z5, tool0;
	MoveL Offs(p0,153.6368,479.1152, 0), v100, z5, tool0;
	MoveL Offs(p0,155.9086,483.2424, 0), v100, z5, tool0;
	MoveL Offs(p0,157.8,487.0, 0), v100, z5, tool0;
	MoveL Offs(p0,161.40000000000003,495.21060000000006, 0), v100, z5, tool0;
	MoveL Offs(p0,164.73600000000005,504.0128000000001, 0), v100, z5, tool0;
	MoveL Offs(p0,167.772,513.2422, 0), v100, z5, tool0;
	MoveL Offs(p0,170.472,522.7344, 0), v100, z5, tool0;
	MoveL Offs(p0,172.8,532.325, 0), v100, z5, tool0;
	MoveL Offs(p0,174.72,541.8496, 0), v100, z5, tool0;
	MoveL Offs(p0,176.196,551.1438, 0), v100, z5, tool0;
	MoveL Offs(p0,177.192,560.0432000000001, 0), v100, z5, tool0;
	MoveL Offs(p0,177.672,568.3834, 0), v100, z5, tool0;
	MoveL Offs(p0,177.6,576.0, 0), v100, z5, tool0;
	MoveL Offs(p0,177.42220000000003,579.2320000000001, 0), v100, z5, tool0;
	MoveL Offs(p0,177.23360000000005,581.8880000000001, 0), v100, z5, tool0;
	MoveL Offs(p0,177.0114,584.028, 0), v100, z5, tool0;
	MoveL Offs(p0,176.7328,585.712, 0), v100, z5, tool0;
	MoveL Offs(p0,176.375,587.0, 0), v100, z5, tool0;
	MoveL Offs(p0,175.9152,587.952, 0), v100, z5, tool0;
	MoveL Offs(p0,175.3306,588.628, 0), v100, z5, tool0;
	MoveL Offs(p0,174.59840000000003,589.0880000000001, 0), v100, z5, tool0;
	MoveL Offs(p0,173.69580000000002,589.392, 0), v100, z5, tool0;
	MoveL Offs(p0,172.6,589.6, 0), v100, z5, tool0;
	MoveL Offs(p0,170.50880000000004,589.7472000000002, 0), v100, z5, tool0;
	MoveL Offs(p0,169.7542,589.5838, 0), v100, z5, tool0;
	MoveL Offs(p0,169.1664,589.1936, 0), v100, z5, tool0;
	MoveL Offs(p0,168.725,588.525, 0), v100, z5, tool0;
	MoveL Offs(p0,168.4096,587.5264, 0), v100, z5, tool0;
	MoveL Offs(p0,168.1998,586.1461999999999, 0), v100, z5, tool0;
	MoveL Offs(p0,168.0752,584.3328, 0), v100, z5, tool0;
	MoveL Offs(p0,168.01540000000003,582.0346000000001, 0), v100, z5, tool0;
	MoveL Offs(p0,168.0,579.2, 0), v100, z5, tool0;
	MoveL Offs(p0,167.9228,575.6126000000002, 0), v100, z5, tool0;
	MoveL Offs(p0,167.69440000000006,572.6528000000002, 0), v100, z5, tool0;
	MoveL Offs(p0,167.31959999999998,570.3242, 0), v100, z5, tool0;
	MoveL Offs(p0,166.8032,568.6304, 0), v100, z5, tool0;
	MoveL Offs(p0,166.15,567.575, 0), v100, z5, tool0;
	MoveL Offs(p0,165.3648,567.1616, 0), v100, z5, tool0;
	MoveL Offs(p0,164.45239999999998,567.3938, 0), v100, z5, tool0;
	MoveL Offs(p0,163.4176,568.2752, 0), v100, z5, tool0;
	MoveL Offs(p0,162.2652,569.8094, 0), v100, z5, tool0;
	MoveL Offs(p0,161.0,572.0, 0), v100, z5, tool0;
	MoveL Offs(p0,159.10400000000004,575.3456000000002, 0), v100, z5, tool0;
	MoveL Offs(p0,158.237,576.4784, 0), v100, z5, tool0;
	MoveL Offs(p0,157.40000000000003,577.2608, 0), v100, z5, tool0;
	MoveL Offs(p0,156.575,577.7, 0), v100, z5, tool0;
	MoveL Offs(p0,155.744,577.8032000000001, 0), v100, z5, tool0;
	MoveL Offs(p0,154.88899999999998,577.5776, 0), v100, z5, tool0;
	MoveL Offs(p0,153.99200000000002,577.0304000000001, 0), v100, z5, tool0;
	MoveL Offs(p0,153.03500000000003,576.1688, 0), v100, z5, tool0;
	MoveL Offs(p0,152.0,575.0, 0), v100, z5, tool0;
	MoveL Offs(p0,149.55519999999999,573.1312, 0), v100, z5, tool0;
	MoveL Offs(p0,148.95,573.15, 0), v100, z5, tool0;
	MoveL Offs(p0,148.28480000000002,573.3728, 0), v100, z5, tool0;
	MoveL Offs(p0,147.52839999999998,573.8044, 0), v100, z5, tool0;
	MoveL Offs(p0,146.64960000000002,574.4496000000001, 0), v100, z5, tool0;
	MoveL Offs(p0,145.6172,575.3131999999999, 0), v100, z5, tool0;
	MoveL Offs(p0,144.4,576.4, 0), v100, z5, tool0;
	MoveL Offs(p0,139.6,581.0, 0), v100, z5, tool0;
	MoveL Offs(p0,136.6,576.6, 0), v100, z5, tool0;
	MoveL Offs(p0,134.9638,574.4598, 0), v100, z5, tool0;
	MoveL Offs(p0,134.4336,573.8576, 0), v100, z5, tool0;
	MoveL Offs(p0,133.925,573.325, 0), v100, z5, tool0;
	MoveL Offs(p0,133.44639999999998,572.8704, 0), v100, z5, tool0;
	MoveL Offs(p0,133.00619999999998,572.5022, 0), v100, z5, tool0;
	MoveL Offs(p0,132.61280000000002,572.2288000000001, 0), v100, z5, tool0;
	MoveL Offs(p0,132.27460000000002,572.0586, 0), v100, z5, tool0;
	MoveL Offs(p0,132.0,572.0, 0), v100, z5, tool0;
	MoveL Offs(p0,130.304,574.2528, 0), v100, z5, tool0;
	MoveL Offs(p0,129.7,575.425, 0), v100, z5, tool0;
	MoveL Offs(p0,129.048,576.7952, 0), v100, z5, tool0;
	MoveL Offs(p0,128.35999999999999,578.3406, 0), v100, z5, tool0;
	MoveL Offs(p0,127.648,580.0384, 0), v100, z5, tool0;
	MoveL Offs(p0,126.924,581.8658, 0), v100, z5, tool0;
	MoveL Offs(p0,126.2,583.8, 0), v100, z5, tool0;
	MoveL Offs(p0,124.63400000000001,587.9076000000002, 0), v100, z5, tool0;
	MoveL Offs(p0,122.96000000000001,591.7968000000002, 0), v100, z5, tool0;
	MoveL Offs(p0,121.21399999999998,595.4172000000001, 0), v100, z5, tool0;
	MoveL Offs(p0,119.43200000000002,598.7184, 0), v100, z5, tool0;
	MoveL Offs(p0,117.65,601.65, 0), v100, z5, tool0;
	MoveL Offs(p0,115.904,604.1616, 0), v100, z5, tool0;
	MoveL Offs(p0,114.22999999999999,606.2028, 0), v100, z5, tool0;
	MoveL Offs(p0,112.66400000000002,607.7232, 0), v100, z5, tool0;
	MoveL Offs(p0,111.242,608.6724, 0), v100, z5, tool0;
	MoveL Offs(p0,110.0,609.0, 0), v100, z5, tool0;
	MoveL Offs(p0,107.99839999999999,609.7452000000001, 0), v100, z5, tool0;
	MoveL Offs(p0,107.1328,610.2864000000001, 0), v100, z5, tool0;
	MoveL Offs(p0,106.2,610.95, 0), v100, z5, tool0;
	MoveL Offs(p0,105.2192,611.7216000000001, 0), v100, z5, tool0;
	MoveL Offs(p0,104.2096,612.5868, 0), v100, z5, tool0;
	MoveL Offs(p0,103.1904,613.5312, 0), v100, z5, tool0;
	MoveL Offs(p0,102.1808,614.5404000000001, 0), v100, z5, tool0;
	MoveL Offs(p0,101.2,615.6, 0), v100, z5, tool0;
	MoveL Offs(p0,97.44640000000001,619.1360000000001, 0), v100, z5, tool0;
	MoveL Offs(p0,95.6146,620.3879999999999, 0), v100, z5, tool0;
	MoveL Offs(p0,93.8752,621.28, 0), v100, z5, tool0;
	MoveL Offs(p0,92.275,621.8, 0), v100, z5, tool0;
	MoveL Offs(p0,90.8608,621.9359999999999, 0), v100, z5, tool0;
	MoveL Offs(p0,89.67940000000002,621.676, 0), v100, z5, tool0;
	MoveL Offs(p0,88.7776,621.008, 0), v100, z5, tool0;
	MoveL Offs(p0,88.2022,619.9200000000001, 0), v100, z5, tool0;
	MoveL Offs(p0,88.0,618.4, 0), v100, z5, tool0;
	MoveL Offs(p0,88.20519999999999,616.1265999999999, 0), v100, z5, tool0;
	MoveL Offs(p0,88.3584,615.1392000000001, 0), v100, z5, tool0;
	MoveL Offs(p0,88.55,614.075, 0), v100, z5, tool0;
	MoveL Offs(p0,88.77759999999999,612.9567999999999, 0), v100, z5, tool0;
	MoveL Offs(p0,89.0388,611.8074, 0), v100, z5, tool0;
	MoveL Offs(p0,89.33120000000001,610.6496000000001, 0), v100, z5, tool0;
	MoveL Offs(p0,89.65240000000001,609.5062, 0), v100, z5, tool0;
	MoveL Offs(p0,90.0,608.4, 0), v100, z5, tool0;
	MoveL Offs(p0,90.74080000000002,605.5232000000002, 0), v100, z5, tool0;
	MoveL Offs(p0,90.9432,604.5138, 0), v100, z5, tool0;
	MoveL Offs(p0,91.03040000000001,603.7696000000001, 0), v100, z5, tool0;
	MoveL Offs(p0,91.0,603.275, 0), v100, z5, tool0;
	MoveL Offs(p0,90.8496,603.0143999999999, 0), v100, z5, tool0;
	MoveL Offs(p0,90.5768,602.9721999999999, 0), v100, z5, tool0;
	MoveL Offs(p0,90.17920000000001,603.1328000000001, 0), v100, z5, tool0;
	MoveL Offs(p0,89.6544,603.4806000000001, 0), v100, z5, tool0;
	MoveL Offs(p0,89.0,604.0, 0), v100, z5, tool0;
	MoveL Offs(p0,86.32160000000002,605.6304000000002, 0), v100, z5, tool0;
	MoveL Offs(p0,85.3244,605.7135999999999, 0), v100, z5, tool0;
	MoveL Offs(p0,84.5648,605.3312000000001, 0), v100, z5, tool0;
	MoveL Offs(p0,84.05,604.5, 0), v100, z5, tool0;
	MoveL Offs(p0,83.7872,603.2367999999999, 0), v100, z5, tool0;
	MoveL Offs(p0,83.7836,601.5584, 0), v100, z5, tool0;
	MoveL Offs(p0,84.04640000000002,599.4816000000001, 0), v100, z5, tool0;
	MoveL Offs(p0,84.58279999999999,597.0232000000001, 0), v100, z5, tool0;
	MoveL Offs(p0,85.4,594.2, 0), v100, z5, tool0;
	MoveL Offs(p0,86.35520000000002,590.9248000000001, 0), v100, z5, tool0;
	MoveL Offs(p0,86.7338,589.3022, 0), v100, z5, tool0;
	MoveL Offs(p0,87.0416,587.7264000000001, 0), v100, z5, tool0;
	MoveL Offs(p0,87.275,586.225, 0), v100, z5, tool0;
	MoveL Offs(p0,87.43039999999999,584.8255999999999, 0), v100, z5, tool0;
	MoveL Offs(p0,87.5042,583.5558, 0), v100, z5, tool0;
	MoveL Offs(p0,87.49280000000002,582.4432, 0), v100, z5, tool0;
	MoveL Offs(p0,87.3926,581.5154, 0), v100, z5, tool0;
	MoveL Offs(p0,87.2,580.8, 0), v100, z5, tool0;
	MoveL Offs(p0,86.12899999999999,578.7983999999999, 0), v100, z5, tool0;
	MoveL Offs(p0,85.808,578.6208000000001, 0), v100, z5, tool0;
	MoveL Offs(p0,85.475,578.7, 0), v100, z5, tool0;
	MoveL Offs(p0,85.112,579.0432, 0), v100, z5, tool0;
	MoveL Offs(p0,84.701,579.6576, 0), v100, z5, tool0;
	MoveL Offs(p0,84.224,580.5504000000001, 0), v100, z5, tool0;
	MoveL Offs(p0,83.663,581.7288000000001, 0), v100, z5, tool0;
	MoveL Offs(p0,83.0,583.2, 0), v100, z5, tool0;
	MoveL Offs(p0,81.90400000000001,585.6486000000001, 0), v100, z5, tool0;
	MoveL Offs(p0,80.88000000000002,587.5968, 0), v100, z5, tool0;
	MoveL Offs(p0,79.904,589.0482, 0), v100, z5, tool0;
	MoveL Offs(p0,78.952,590.0064, 0), v100, z5, tool0;
	MoveL Offs(p0,78.0,590.475, 0), v100, z5, tool0;
	MoveL Offs(p0,77.024,590.4576, 0), v100, z5, tool0;
	MoveL Offs(p0,76.0,589.9577999999999, 0), v100, z5, tool0;
	MoveL Offs(p0,74.90400000000001,588.9792, 0), v100, z5, tool0;
	MoveL Offs(p0,73.712,587.5254, 0), v100, z5, tool0;
	MoveL Offs(p0,72.4,585.6, 0), v100, z5, tool0;
	MoveL Offs(p0,68.4,579.4, 0), v100, z5, tool0;
	MoveL Offs(p0,65.2,585.6, 0), v100, z5, tool0;
	MoveL Offs(p0,64.08640000000003,587.648, 0), v100, z5, tool0;
	MoveL Offs(p0,63.52059999999999,588.5699999999999, 0), v100, z5, tool0;
	MoveL Offs(p0,62.96320000000001,589.4080000000001, 0), v100, z5, tool0;
	MoveL Offs(p0,62.425,590.15, 0), v100, z5, tool0;
	MoveL Offs(p0,61.9168,590.784, 0), v100, z5, tool0;
	MoveL Offs(p0,61.449400000000004,591.298, 0), v100, z5, tool0;
	MoveL Offs(p0,61.0336,591.6800000000001, 0), v100, z5, tool0;
	MoveL Offs(p0,60.6802,591.918, 0), v100, z5, tool0;
	MoveL Offs(p0,60.4,592.0, 0), v100, z5, tool0;
	MoveL Offs(p0,58.175,589.8, 0), v100, z5, tool0;
	MoveL Offs(p0,57.606399999999994,588.9327999999999, 0), v100, z5, tool0;
	MoveL Offs(p0,57.01619999999999,587.9624, 0), v100, z5, tool0;
	MoveL Offs(p0,56.412800000000004,586.9056, 0), v100, z5, tool0;
	MoveL Offs(p0,55.80460000000001,585.7792000000001, 0), v100, z5, tool0;
	MoveL Offs(p0,55.2,584.6, 0), v100, z5, tool0;
	MoveL Offs(p0,53.47840000000002,581.1904000000002, 0), v100, z5, tool0;
	MoveL Offs(p0,52.8096,580.0495999999999, 0), v100, z5, tool0;
	MoveL Offs(p0,52.2272,579.2592000000002, 0), v100, z5, tool0;
	MoveL Offs(p0,51.7,578.8, 0), v100, z5, tool0;
	MoveL Offs(p0,51.1968,578.6528000000001, 0), v100, z5, tool0;
	MoveL Offs(p0,50.686400000000006,578.7983999999999, 0), v100, z5, tool0;
	MoveL Offs(p0,50.137600000000006,579.2176000000001, 0), v100, z5, tool0;
	MoveL Offs(p0,49.5192,579.8912, 0), v100, z5, tool0;
	MoveL Offs(p0,48.8,580.8, 0), v100, z5, tool0;
	MoveL Offs(p0,47.113600000000005,583.4304, 0), v100, z5, tool0;
	MoveL Offs(p0,46.725,584.1, 0), v100, z5, tool0;
	MoveL Offs(p0,46.3664,584.7456, 0), v100, z5, tool0;
	MoveL Offs(p0,46.0462,585.3527999999999, 0), v100, z5, tool0;
	MoveL Offs(p0,45.772800000000004,585.9072, 0), v100, z5, tool0;
	MoveL Offs(p0,45.55460000000001,586.3944, 0), v100, z5, tool0;
	MoveL Offs(p0,45.4,586.8, 0), v100, z5, tool0;
	MoveL Offs(p0,43.2776,587.5826, 0), v100, z5, tool0;
	MoveL Offs(p0,42.78240000000001,587.2864000000002, 0), v100, z5, tool0;
	MoveL Offs(p0,42.2248,586.8918000000001, 0), v100, z5, tool0;
	MoveL Offs(p0,41.6,586.4, 0), v100, z5, tool0;
	MoveL Offs(p0,39.216,585.0975999999999, 0), v100, z5, tool0;
	MoveL Offs(p0,38.8,585.225, 0), v100, z5, tool0;
	MoveL Offs(p0,38.432,585.5504, 0), v100, z5, tool0;
	MoveL Offs(p0,38.1,586.0822000000001, 0), v100, z5, tool0;
	MoveL Offs(p0,37.79200000000001,586.8288, 0), v100, z5, tool0;
	MoveL Offs(p0,37.496,587.7986, 0), v100, z5, tool0;
	MoveL Offs(p0,37.2,589.0, 0), v100, z5, tool0;
	MoveL Offs(p0,36.2046,591.5793999999999, 0), v100, z5, tool0;
	MoveL Offs(p0,35.74720000000001,592.2288000000001, 0), v100, z5, tool0;
	MoveL Offs(p0,35.225,592.775, 0), v100, z5, tool0;
	MoveL Offs(p0,34.6368,593.2192, 0), v100, z5, tool0;
	MoveL Offs(p0,33.9814,593.5626, 0), v100, z5, tool0;
	MoveL Offs(p0,33.257600000000004,593.8064, 0), v100, z5, tool0;
	MoveL Offs(p0,32.4642,593.9518, 0), v100, z5, tool0;
	MoveL Offs(p0,31.6,594.0, 0), v100, z5, tool0;
	MoveL Offs(p0,28.961199999999998,593.4707999999998, 0), v100, z5, tool0;
	MoveL Offs(p0,28.4704,592.8416, 0), v100, z5, tool0;
	MoveL Offs(p0,28.15,591.85, 0), v100, z5, tool0;
	MoveL Offs(p0,27.985599999999998,590.4143999999999, 0), v100, z5, tool0;
	MoveL Offs(p0,27.962799999999998,588.4531999999999, 0), v100, z5, tool0;
	MoveL Offs(p0,28.067200000000003,585.8848, 0), v100, z5, tool0;
	MoveL Offs(p0,28.284400000000005,582.6276, 0), v100, z5, tool0;
	MoveL Offs(p0,28.6,578.6, 0), v100, z5, tool0;
	MoveL Offs(p0,29.609400000000004,569.6076000000002, 0), v100, z5, tool0;
	MoveL Offs(p0,31.179200000000016,560.3248000000002, 0), v100, z5, tool0;
	MoveL Offs(p0,33.281800000000004,550.8331999999999, 0), v100, z5, tool0;
	MoveL Offs(p0,35.8896,541.2144000000001, 0), v100, z5, tool0;
	MoveL Offs(p0,38.975,531.55, 0), v100, z5, tool0;
	MoveL Offs(p0,42.510400000000004,521.9216, 0), v100, z5, tool0;
	MoveL Offs(p0,46.4682,512.4108, 0), v100, z5, tool0;
	MoveL Offs(p0,50.820800000000006,503.0992, 0), v100, z5, tool0;
	MoveL Offs(p0,55.540600000000005,494.0684, 0), v100, z5, tool0;
	MoveL Offs(p0,60.6,485.4, 0), v100, z5, tool0;
	MoveL Offs(p0,64.59220000000002,478.9264, 0), v100, z5, tool0;
	MoveL Offs(p0,67.72160000000002,473.7872000000002, 0), v100, z5, tool0;
	MoveL Offs(p0,70.0374,469.80480000000006, 0), v100, z5, tool0;
	MoveL Offs(p0,71.5888,466.8016000000001, 0), v100, z5, tool0;
	MoveL Offs(p0,72.425,464.6, 0), v100, z5, tool0;
	MoveL Offs(p0,72.5952,463.0224, 0), v100, z5, tool0;
	MoveL Offs(p0,72.1486,461.8912, 0), v100, z5, tool0;
	MoveL Offs(p0,71.1344,461.02880000000005, 0), v100, z5, tool0;
	MoveL Offs(p0,69.6018,460.2576, 0), v100, z5, tool0;
	MoveL Offs(p0,67.6,459.4, 0), v100, z5, tool0;
	MoveL Offs(p0,63.1792,457.0418000000001, 0), v100, z5, tool0;
	MoveL Offs(p0,58.94560000000001,453.85440000000017, 0), v100, z5, tool0;
	MoveL Offs(p0,54.9424,449.90860000000004, 0), v100, z5, tool0;
	MoveL Offs(p0,51.212800000000016,445.27520000000004, 0), v100, z5, tool0;
	MoveL Offs(p0,47.8,440.025, 0), v100, z5, tool0;
	MoveL Offs(p0,44.7472,434.22880000000004, 0), v100, z5, tool0;
	MoveL Offs(p0,42.09759999999999,427.95739999999995, 0), v100, z5, tool0;
	MoveL Offs(p0,39.894400000000005,421.2816000000001, 0), v100, z5, tool0;
	MoveL Offs(p0,38.1808,414.2722, 0), v100, z5, tool0;
	MoveL Offs(p0,37.0,407.0, 0), v100, z5, tool0;
	MoveL Offs(p0,36.6266,404.45180000000005, 0), v100, z5, tool0;
	MoveL Offs(p0,36.22080000000001,402.19040000000007, 0), v100, z5, tool0;
	MoveL Offs(p0,35.77420000000001,400.19059999999996, 0), v100, z5, tool0;
	MoveL Offs(p0,35.2784,398.42719999999997, 0), v100, z5, tool0;
	MoveL Offs(p0,34.725,396.875, 0), v100, z5, tool0;
	MoveL Offs(p0,34.105599999999995,395.5088, 0), v100, z5, tool0;
	MoveL Offs(p0,33.4118,394.3034, 0), v100, z5, tool0;
	MoveL Offs(p0,32.635200000000005,393.2336, 0), v100, z5, tool0;
	MoveL Offs(p0,31.767400000000002,392.2742, 0), v100, z5, tool0;
	MoveL Offs(p0,30.8,391.4, 0), v100, z5, tool0;
	MoveL Offs(p0,27.811999999999994,388.04479999999995, 0), v100, z5, tool0;
	MoveL Offs(p0,26.592000000000002,386.3376, 0), v100, z5, tool0;
	MoveL Offs(p0,25.3,384.4, 0), v100, z5, tool0;
	MoveL Offs(p0,23.96,382.2704, 0), v100, z5, tool0;
	MoveL Offs(p0,22.595999999999997,379.9871999999999, 0), v100, z5, tool0;
	MoveL Offs(p0,21.232000000000003,377.5888, 0), v100, z5, tool0;
	MoveL Offs(p0,19.892000000000003,375.1136, 0), v100, z5, tool0;
	MoveL Offs(p0,18.6,372.6, 0), v100, z5, tool0;
	MoveL Offs(p0,16.6372,368.52880000000005, 0), v100, z5, tool0;
	MoveL Offs(p0,15.041600000000006,365.0624000000001, 0), v100, z5, tool0;
	MoveL Offs(p0,13.7724,362.00159999999994, 0), v100, z5, tool0;
	MoveL Offs(p0,12.788800000000002,359.14720000000005, 0), v100, z5, tool0;
	MoveL Offs(p0,12.05,356.3, 0), v100, z5, tool0;
	MoveL Offs(p0,11.5152,353.2608, 0), v100, z5, tool0;
	MoveL Offs(p0,11.143600000000001,349.8304, 0), v100, z5, tool0;
	MoveL Offs(p0,10.894400000000001,345.80960000000005, 0), v100, z5, tool0;
	MoveL Offs(p0,10.7268,340.99920000000003, 0), v100, z5, tool0;
	MoveL Offs(p0,10.6,335.2, 0), v100, z5, tool0;
	MoveL Offs(p0,10.514200000000002,330.09720000000004, 0), v100, z5, tool0;
	MoveL Offs(p0,10.369600000000002,325.6496000000001, 0), v100, z5, tool0;
	MoveL Offs(p0,10.155399999999998,321.7684, 0), v100, z5, tool0;
	MoveL Offs(p0,9.860800000000001,318.3648, 0), v100, z5, tool0;
	MoveL Offs(p0,9.475,315.35, 0), v100, z5, tool0;
	MoveL Offs(p0,8.9872,312.6352, 0), v100, z5, tool0;
	MoveL Offs(p0,8.3866,310.1316, 0), v100, z5, tool0;
	MoveL Offs(p0,7.662400000000001,307.7504, 0), v100, z5, tool0;
	MoveL Offs(p0,6.8038,305.4028, 0), v100, z5, tool0;
	MoveL Offs(p0,5.8,303.0, 0), v100, z5, tool0;
	MoveL Offs(p0,3.935,297.94700000000006, 0), v100, z5, tool0;
	MoveL Offs(p0,2.4240000000000004,291.92800000000005, 0), v100, z5, tool0;
	MoveL Offs(p0,1.2729999999999992,285.15299999999996, 0), v100, z5, tool0;
	MoveL Offs(p0,0.4879999999999998,277.832, 0), v100, z5, tool0;
	MoveL Offs(p0,0.075,270.175, 0), v100, z5, tool0;
	MoveL Offs(p0,0.040000000000000216,262.392, 0), v100, z5, tool0;
	MoveL Offs(p0,0.38900000000000023,254.69299999999998, 0), v100, z5, tool0;
	MoveL Offs(p0,1.1280000000000003,247.288, 0), v100, z5, tool0;
	MoveL Offs(p0,2.263000000000001,240.387, 0), v100, z5, tool0;
	MoveL Offs(p0,3.8,234.2, 0), v100, z5, tool0;
	MoveL Offs(p0,4.500800000000001,231.844, 0), v100, z5, tool0;
	MoveL Offs(p0,5.158400000000001,229.36800000000008, 0), v100, z5, tool0;
	MoveL Offs(p0,5.765600000000001,226.82, 0), v100, z5, tool0;
	MoveL Offs(p0,6.315200000000002,224.248, 0), v100, z5, tool0;
	MoveL Offs(p0,6.8,221.7, 0), v100, z5, tool0;
	MoveL Offs(p0,7.212800000000001,219.224, 0), v100, z5, tool0;
	MoveL Offs(p0,7.5464,216.868, 0), v100, z5, tool0;
	MoveL Offs(p0,7.7936000000000005,214.68, 0), v100, z5, tool0;
	MoveL Offs(p0,7.9472000000000005,212.708, 0), v100, z5, tool0;
	MoveL Offs(p0,8.0,211.0, 0), v100, z5, tool0;
	MoveL Offs(p0,8.2306,207.497, 0), v100, z5, tool0;
	MoveL Offs(p0,8.884800000000002,203.23200000000003, 0), v100, z5, tool0;
	MoveL Offs(p0,9.906200000000002,198.391, 0), v100, z5, tool0;
	MoveL Offs(p0,11.238400000000002,193.16000000000003, 0), v100, z5, tool0;
	MoveL Offs(p0,12.825,187.725, 0), v100, z5, tool0;
	MoveL Offs(p0,14.609600000000004,182.272, 0), v100, z5, tool0;
	MoveL Offs(p0,16.535800000000002,176.987, 0), v100, z5, tool0;
	MoveL Offs(p0,18.547200000000004,172.05599999999998, 0), v100, z5, tool0;
	MoveL Offs(p0,20.587400000000002,167.66500000000002, 0), v100, z5, tool0;
	MoveL Offs(p0,22.6,164.0, 0), v100, z5, tool0;
	MoveL Offs(p0,24.26880000000001,161.31200000000007, 0), v100, z5, tool0;
	MoveL Offs(p0,25.3252,159.71599999999998, 0), v100, z5, tool0;
	MoveL Offs(p0,26.494400000000002,158.00000000000003, 0), v100, z5, tool0;
	MoveL Offs(p0,27.75,156.2, 0), v100, z5, tool0;
	MoveL Offs(p0,29.0656,154.352, 0), v100, z5, tool0;
	MoveL Offs(p0,30.414799999999996,152.49200000000002, 0), v100, z5, tool0;
	MoveL Offs(p0,31.771200000000004,150.656, 0), v100, z5, tool0;
	MoveL Offs(p0,33.1084,148.88000000000002, 0), v100, z5, tool0;
	MoveL Offs(p0,34.4,147.2, 0), v100, z5, tool0;
	MoveL Offs(p0,36.80320000000001,143.94720000000004, 0), v100, z5, tool0;
	MoveL Offs(p0,37.8938,142.3508, 0), v100, z5, tool0;
	MoveL Offs(p0,38.889599999999994,140.8096, 0), v100, z5, tool0;
	MoveL Offs(p0,39.775,139.35, 0), v100, z5, tool0;
	MoveL Offs(p0,40.53439999999999,137.9984, 0), v100, z5, tool0;
	MoveL Offs(p0,41.15220000000001,136.78119999999998, 0), v100, z5, tool0;
	MoveL Offs(p0,41.61280000000001,135.72480000000002, 0), v100, z5, tool0;
	MoveL Offs(p0,41.900600000000004,134.8556, 0), v100, z5, tool0;
	MoveL Offs(p0,42.0,134.2, 0), v100, z5, tool0;
	MoveL Offs(p0,42.65339999999999,131.3164, 0), v100, z5, tool0;
	MoveL Offs(p0,43.13280000000001,129.87680000000003, 0), v100, z5, tool0;
	MoveL Offs(p0,43.725,128.25, 0), v100, z5, tool0;
	MoveL Offs(p0,44.419200000000004,126.4672, 0), v100, z5, tool0;
	MoveL Offs(p0,45.2046,124.5596, 0), v100, z5, tool0;
	MoveL Offs(p0,46.07040000000001,122.55840000000003, 0), v100, z5, tool0;
	MoveL Offs(p0,47.00580000000001,120.49480000000001, 0), v100, z5, tool0;
	MoveL Offs(p0,48.0,118.4, 0), v100, z5, tool0;
	MoveL Offs(p0,50.463800000000006,113.75280000000001, 0), v100, z5, tool0;
	MoveL Offs(p0,53.47840000000001,108.99040000000005, 0), v100, z5, tool0;
	MoveL Offs(p0,56.95859999999999,104.20159999999998, 0), v100, z5, tool0;
	MoveL Offs(p0,60.8192,99.4752, 0), v100, z5, tool0;
	MoveL Offs(p0,64.975,94.9, 0), v100, z5, tool0;
	MoveL Offs(p0,69.3408,90.56479999999999, 0), v100, z5, tool0;
	MoveL Offs(p0,73.8314,86.55839999999999, 0), v100, z5, tool0;
	MoveL Offs(p0,78.36160000000001,82.96960000000001, 0), v100, z5, tool0;
	MoveL Offs(p0,82.84620000000001,79.8872, 0), v100, z5, tool0;
	MoveL Offs(p0,87.2,77.4, 0), v100, z5, tool0;
	MoveL Offs(p0,90.50560000000003,75.55200000000002, 0), v100, z5, tool0;
	MoveL Offs(p0,92.08340000000001,74.52899999999998, 0), v100, z5, tool0;
	MoveL Offs(p0,93.58080000000001,73.46400000000001, 0), v100, z5, tool0;
	MoveL Offs(p0,94.975,72.375, 0), v100, z5, tool0;
	MoveL Offs(p0,96.24319999999999,71.28, 0), v100, z5, tool0;
	MoveL Offs(p0,97.3626,70.197, 0), v100, z5, tool0;
	MoveL Offs(p0,98.3104,69.144, 0), v100, z5, tool0;
	MoveL Offs(p0,99.0638,68.139, 0), v100, z5, tool0;
	MoveL Offs(p0,99.6,67.2, 0), v100, z5, tool0;
	MoveL Offs(p0,102.99340000000002,61.2626, 0), v100, z5, tool0;
	MoveL Offs(p0,107.76320000000003,55.29280000000002, 0), v100, z5, tool0;
	MoveL Offs(p0,113.71379999999999,49.414199999999994, 0), v100, z5, tool0;
	MoveL Offs(p0,120.6496,43.7504, 0), v100, z5, tool0;
	MoveL Offs(p0,128.375,38.425, 0), v100, z5, tool0;
	MoveL Offs(p0,136.6944,33.5616, 0), v100, z5, tool0;
	MoveL Offs(p0,145.4122,29.283799999999996, 0), v100, z5, tool0;
	MoveL Offs(p0,154.33280000000002,25.7152, 0), v100, z5, tool0;
	MoveL Offs(p0,163.2606,22.979400000000002, 0), v100, z5, tool0;
	MoveL Offs(p0,172.0,21.2, 0), v100, z5, tool0;
	MoveL Offs(p0,175.58240000000004,20.384000000000007, 0), v100, z5, tool0;
	MoveL Offs(p0,177.7366,19.750999999999998, 0), v100, z5, tool0;
	MoveL Offs(p0,180.0672,18.992, 0), v100, z5, tool0;
	MoveL Offs(p0,182.525,18.125, 0), v100, z5, tool0;
	MoveL Offs(p0,185.06080000000003,17.168, 0), v100, z5, tool0;
	MoveL Offs(p0,187.62539999999998,16.139, 0), v100, z5, tool0;
	MoveL Offs(p0,190.1696,15.056000000000001, 0), v100, z5, tool0;
	MoveL Offs(p0,192.6442,13.937000000000001, 0), v100, z5, tool0;
	MoveL Offs(p0,195.0,12.8, 0), v100, z5, tool0;
	MoveL Offs(p0,201.3864,9.8016, 0), v100, z5, tool0;
	MoveL Offs(p0,207.42720000000003,7.268800000000003, 0), v100, z5, tool0;
	MoveL Offs(p0,213.24479999999994,5.1751999999999985, 0), v100, z5, tool0;
	MoveL Offs(p0,218.9616,3.4943999999999997, 0), v100, z5, tool0;
	MoveL Offs(p0,224.7,2.2, 0), v100, z5, tool0;
	MoveL Offs(p0,230.5824,1.2655999999999994, 0), v100, z5, tool0;
	MoveL Offs(p0,236.7312,0.6647999999999997, 0), v100, z5, tool0;
	MoveL Offs(p0,243.2688,0.3711999999999999, 0), v100, z5, tool0;
	MoveL Offs(p0,250.3176,0.35840000000000005, 0), v100, z5, tool0;
	MoveL Offs(p0,258.0,0.6, 0), v100, z5, tool0;
	MoveL Offs(p0,262.10940000000005,0.8150000000000002, 0), v100, z5, tool0;
	MoveL Offs(p0,266.13120000000004,1.0960000000000003, 0), v100, z5, tool0;
	MoveL Offs(p0,270.02579999999995,1.437, 0), v100, z5, tool0;
	MoveL Offs(p0,273.75360000000006,1.832, 0), v100, z5, tool0;
	MoveL Offs(p0,277.275,2.275, 0), v100, z5, tool0;
	MoveL Offs(p0,280.55039999999997,2.7600000000000002, 0), v100, z5, tool0;
	MoveL Offs(p0,283.5402,3.281, 0), v100, z5, tool0;
	MoveL Offs(p0,286.20480000000003,3.8320000000000007, 0), v100, z5, tool0;
	MoveL Offs(p0,288.5046,4.407, 0), v100, z5, tool0;
	MoveL Offs(p0,290.4,5.0, 0), v100, z5, tool0;
	MoveL Offs(p0,292.74260000000004,5.8112, 0), v100, z5, tool0;
	MoveL Offs(p0,294.90880000000004,6.449600000000001, 0), v100, z5, tool0;
	MoveL Offs(p0,296.98619999999994,6.9224000000000006, 0), v100, z5, tool0;
	MoveL Offs(p0,299.0624,7.236800000000001, 0), v100, z5, tool0;
	MoveL Offs(p0,301.225,7.4, 0), v100, z5, tool0;
	MoveL Offs(p0,303.5616,7.419200000000001, 0), v100, z5, tool0;
	MoveL Offs(p0,306.1598,7.301599999999999, 0), v100, z5, tool0;
	MoveL Offs(p0,309.10720000000003,7.054400000000001, 0), v100, z5, tool0;
	MoveL Offs(p0,312.4914,6.6848, 0), v100, z5, tool0;
	MoveL Offs(p0,316.4,6.2, 0), v100, z5, tool0;
	MoveL Offs(p0,332.30060000000003,5.133800000000001, 0), v100, z5, tool0;
	MoveL Offs(p0,348.3728000000001,6.046400000000001, 0), v100, z5, tool0;
	MoveL Offs(p0,364.3322,8.8046, 0), v100, z5, tool0;
	MoveL Offs(p0,379.8944,13.275200000000002, 0), v100, z5, tool0;
	MoveL Offs(p0,394.775,19.325, 0), v100, z5, tool0;
	MoveL Offs(p0,408.68960000000004,26.82080000000001, 0), v100, z5, tool0;
	MoveL Offs(p0,421.35380000000004,35.62940000000001, 0), v100, z5, tool0;
	MoveL Offs(p0,432.4832,45.61760000000001, 0), v100, z5, tool0;
	MoveL Offs(p0,441.7934,56.65220000000001, 0), v100, z5, tool0;
	MoveL Offs(p0,449.0,68.6, 0), v100, z5, tool0;
	MoveL Offs(p0,450.2706,71.10640000000001, 0), v100, z5, tool0;
	MoveL Offs(p0,451.48480000000006,73.26720000000002, 0), v100, z5, tool0;
	MoveL Offs(p0,452.70619999999997,75.14479999999999, 0), v100, z5, tool0;
	MoveL Offs(p0,453.99840000000006,76.80160000000001, 0), v100, z5, tool0;
	MoveL Offs(p0,455.425,78.3, 0), v100, z5, tool0;
	MoveL Offs(p0,457.0496,79.7024, 0), v100, z5, tool0;
	MoveL Offs(p0,458.93580000000003,81.0712, 0), v100, z5, tool0;
	MoveL Offs(p0,461.1472,82.46880000000002, 0), v100, z5, tool0;
	MoveL Offs(p0,463.7474,83.9576, 0), v100, z5, tool0;
	MoveL Offs(p0,466.8,85.6, 0), v100, z5, tool0;
	MoveL Offs(p0,475.22660000000013,90.73440000000002, 0), v100, z5, tool0;
	MoveL Offs(p0,483.1648,97.03520000000002, 0), v100, z5, tool0;
	MoveL Offs(p0,490.5221999999999,104.34880000000001, 0), v100, z5, tool0;
	MoveL Offs(p0,497.20640000000003,112.5216, 0), v100, z5, tool0;
	MoveL Offs(p0,503.125,121.4, 0), v100, z5, tool0;
	MoveL Offs(p0,508.18559999999997,130.8304, 0), v100, z5, tool0;
	MoveL Offs(p0,512.2958000000001,140.6592, 0), v100, z5, tool0;
	MoveL Offs(p0,515.3632,150.73280000000003, 0), v100, z5, tool0;
	MoveL Offs(p0,517.2954,160.8976, 0), v100, z5, tool0;
	MoveL Offs(p0,518.0,171.0, 0), v100, z5, tool0;
	MoveL Offs(p0,518.2288000000001,174.46560000000002, 0), v100, z5, tool0;
	MoveL Offs(p0,518.5292000000001,176.1354, 0), v100, z5, tool0;
	MoveL Offs(p0,518.9664,177.79680000000002, 0), v100, z5, tool0;
	MoveL Offs(p0,519.55,179.475, 0), v100, z5, tool0;
	MoveL Offs(p0,520.2896000000001,181.1952, 0), v100, z5, tool0;
	MoveL Offs(p0,521.1948,182.9826, 0), v100, z5, tool0;
	MoveL Offs(p0,522.2752,184.86240000000004, 0), v100, z5, tool0;
	MoveL Offs(p0,523.5404000000001,186.8598, 0), v100, z5, tool0;
	MoveL Offs(p0,525.0,189.0, 0), v100, z5, tool0;
	MoveL Offs(p0,528.6604000000001,194.84220000000002, 0), v100, z5, tool0;
	MoveL Offs(p0,531.9392,201.46560000000005, 0), v100, z5, tool0;
	MoveL Offs(p0,534.8028,208.7154, 0), v100, z5, tool0;
	MoveL Offs(p0,537.2176000000001,216.43680000000003, 0), v100, z5, tool0;
	MoveL Offs(p0,539.15,224.475, 0), v100, z5, tool0;
	MoveL Offs(p0,540.5664,232.6752, 0), v100, z5, tool0;
	MoveL Offs(p0,541.4332,240.8826, 0), v100, z5, tool0;
	MoveL Offs(p0,541.7168,248.9424, 0), v100, z5, tool0;
	MoveL Offs(p0,541.3836,256.6998, 0), v100, z5, tool0;
	MoveL Offs(p0,540.4,264.0, 0), v100, z5, tool0;
	MoveL Offs(p0,539.7552000000003,267.49120000000005, 0), v100, z5, tool0;
	MoveL Offs(p0,539.4927999999999,269.11379999999997, 0), v100, z5, tool0;
	MoveL Offs(p0,539.2736,270.6176, 0), v100, z5, tool0;
	MoveL Offs(p0,539.1,271.975, 0), v100, z5, tool0;
	MoveL Offs(p0,538.9744,273.1584, 0), v100, z5, tool0;
	MoveL Offs(p0,538.8992000000001,274.1402, 0), v100, z5, tool0;
	MoveL Offs(p0,538.8768,274.8928, 0), v100, z5, tool0;
	MoveL Offs(p0,538.9096,275.3886, 0), v100, z5, tool0;
	MoveL Offs(p0,539.0,275.6, 0), v100, z5, tool0;
	MoveL Offs(p0,542.1232,273.38559999999995, 0), v100, z5, tool0;
	MoveL Offs(p0,543.6,272.1, 0), v100, z5, tool0;
	MoveL Offs(p0,545.2927999999999,270.57439999999997, 0), v100, z5, tool0;
	MoveL Offs(p0,547.1704,268.8352, 0), v100, z5, tool0;
	MoveL Offs(p0,549.2016000000001,266.90880000000004, 0), v100, z5, tool0;
	MoveL Offs(p0,551.3552,264.82160000000005, 0), v100, z5, tool0;
	MoveL Offs(p0,553.6,262.6, 0), v100, z5, tool0;
	MoveL Offs(p0,558.8454000000002,257.2252000000001, 0), v100, z5, tool0;
	MoveL Offs(p0,563.8832000000002,251.5696000000001, 0), v100, z5, tool0;
	MoveL Offs(p0,568.6858,245.6764, 0), v100, z5, tool0;
	MoveL Offs(p0,573.2256,239.58880000000005, 0), v100, z5, tool0;
	MoveL Offs(p0,577.475,233.35, 0), v100, z5, tool0;
	MoveL Offs(p0,581.4064000000001,227.00320000000002, 0), v100, z5, tool0;
	MoveL Offs(p0,584.9922,220.59160000000003, 0), v100, z5, tool0;
	MoveL Offs(p0,588.2048000000001,214.15840000000003, 0), v100, z5, tool0;
	MoveL Offs(p0,591.0166,207.74679999999998, 0), v100, z5, tool0;
	MoveL Offs(p0,593.4,201.4, 0), v100, z5, tool0;
	MoveL Offs(p0,594.7718000000001,197.342, 0), v100, z5, tool0;
	MoveL Offs(p0,595.9024000000002,193.70400000000006, 0), v100, z5, tool0;
	MoveL Offs(p0,596.8145999999999,190.32999999999998, 0), v100, z5, tool0;
	MoveL Offs(p0,597.5312,187.06400000000002, 0), v100, z5, tool0;
	MoveL Offs(p0,598.075,183.75, 0), v100, z5, tool0;
	MoveL Offs(p0,598.4688,180.23200000000003, 0), v100, z5, tool0;
	MoveL Offs(p0,598.7354,176.35399999999998, 0), v100, z5, tool0;
	MoveL Offs(p0,598.8976,171.96, 0), v100, z5, tool0;
	MoveL Offs(p0,598.9782000000001,166.894, 0), v100, z5, tool0;
	MoveL Offs(p0,599.0,161.0, 0), v100, z5, tool0;
	MoveL Offs(p0,598.9738000000001,155.3588, 0), v100, z5, tool0;
	MoveL Offs(p0,598.8864000000001,150.47840000000002, 0), v100, z5, tool0;
	MoveL Offs(p0,598.7246,146.2436, 0), v100, z5, tool0;
	MoveL Offs(p0,598.4752000000001,142.5392, 0), v100, z5, tool0;
	MoveL Offs(p0,598.125,139.25, 0), v100, z5, tool0;
	MoveL Offs(p0,597.6608,136.26079999999996, 0), v100, z5, tool0;
	MoveL Offs(p0,597.0694,133.45639999999997, 0), v100, z5, tool0;
	MoveL Offs(p0,596.3376000000001,130.7216, 0), v100, z5, tool0;
	MoveL Offs(p0,595.4522,127.94120000000001, 0), v100, z5, tool0;
	MoveL Offs(p0,594.4,125.0, 0), v100, z5, tool0;
	MoveL Offs(p0,592.4878,120.29220000000002, 0), v100, z5, tool0;
	MoveL Offs(p0,590.3584000000002,115.77760000000004, 0), v100, z5, tool0;
	MoveL Offs(p0,588.0226,111.4694, 0), v100, z5, tool0;
	MoveL Offs(p0,585.4912000000002,107.3808, 0), v100, z5, tool0;
	MoveL Offs(p0,582.775,103.525, 0), v100, z5, tool0;
	MoveL Offs(p0,579.8848,99.9152, 0), v100, z5, tool0;
	MoveL Offs(p0,576.8314,96.5646, 0), v100, z5, tool0;
	MoveL Offs(p0,573.6256000000001,93.4864, 0), v100, z5, tool0;
	MoveL Offs(p0,570.2782,90.69380000000001, 0), v100, z5, tool0;
	MoveL Offs(p0,566.8,88.2, 0), v100, z5, tool0;
	MoveL Offs(p0,559.5890000000002,83.9462, 0), v100, z5, tool0;
	MoveL Offs(p0,552.72,80.90560000000002, 0), v100, z5, tool0;
	MoveL Offs(p0,546.199,79.07939999999999, 0), v100, z5, tool0;
	MoveL Offs(p0,540.0319999999999,78.4688, 0), v100, z5, tool0;
	MoveL Offs(p0,534.225,79.075, 0), v100, z5, tool0;
	MoveL Offs(p0,528.784,80.89920000000001, 0), v100, z5, tool0;
	MoveL Offs(p0,523.7149999999999,83.9426, 0), v100, z5, tool0;
	MoveL Offs(p0,519.024,88.2064, 0), v100, z5, tool0;
	MoveL Offs(p0,514.717,93.6918, 0), v100, z5, tool0;
	MoveL Offs(p0,510.8,100.4, 0), v100, z5, tool0;
	MoveL Offs(p0,508.7744000000001,104.08320000000003, 0), v100, z5, tool0;
	MoveL Offs(p0,507.85159999999996,105.5498, 0), v100, z5, tool0;
	MoveL Offs(p0,506.97919999999993,106.7776, 0), v100, z5, tool0;
	MoveL Offs(p0,506.15,107.775, 0), v100, z5, tool0;
	MoveL Offs(p0,505.3567999999999,108.5504, 0), v100, z5, tool0;
	MoveL Offs(p0,504.5924,109.1122, 0), v100, z5, tool0;
	MoveL Offs(p0,503.8496,109.46880000000002, 0), v100, z5, tool0;
	MoveL Offs(p0,503.12120000000004,109.6286, 0), v100, z5, tool0;
	MoveL Offs(p0,502.4,109.6, 0), v100, z5, tool0;
	MoveL Offs(p0,499.9616000000001,107.22240000000004, 0), v100, z5, tool0;
	MoveL Offs(p0,499.32739999999995,104.97759999999998, 0), v100, z5, tool0;
	MoveL Offs(p0,499.0688,102.1952, 0), v100, z5, tool0;
	MoveL Offs(p0,499.175,99.0, 0), v100, z5, tool0;
	MoveL Offs(p0,499.6352,95.51679999999999, 0), v100, z5, tool0;
	MoveL Offs(p0,500.43860000000006,91.87039999999999, 0), v100, z5, tool0;
	MoveL Offs(p0,501.5744000000001,88.1856, 0), v100, z5, tool0;
	MoveL Offs(p0,503.03180000000003,84.58720000000001, 0), v100, z5, tool0;
	MoveL Offs(p0,504.8,81.2, 0), v100, z5, tool0;
	MoveL Offs(p0,507.94620000000015,76.45540000000001, 0), v100, z5, tool0;
	MoveL Offs(p0,511.48960000000017,72.30720000000002, 0), v100, z5, tool0;
	MoveL Offs(p0,515.4073999999999,68.7638, 0), v100, z5, tool0;
	MoveL Offs(p0,519.6768,65.8336, 0), v100, z5, tool0;
	MoveL Offs(p0,524.275,63.525, 0), v100, z5, tool0;
	MoveL Offs(p0,529.1792,61.846399999999996, 0), v100, z5, tool0;
	MoveL Offs(p0,534.3666000000001,60.806200000000004, 0), v100, z5, tool0;
	MoveL Offs(p0,539.8144,60.412800000000004, 0), v100, z5, tool0;
	MoveL Offs(p0,545.4998,60.67460000000001, 0), v100, z5, tool0;
	MoveL Offs(p0,551.4,61.6, 0), v100, z5, tool0;
	MoveL Offs(p0,561.6002000000001,64.35460000000002, 0), v100, z5, tool0;
	MoveL Offs(p0,571.1776000000002,68.1568, 0), v100, z5, tool0;
	MoveL Offs(p0,580.0973999999999,72.97420000000001, 0), v100, z5, tool0;
	MoveL Offs(p0,588.3248000000001,78.7744, 0), v100, z5, tool0;
	MoveL Offs(p0,595.825,85.525, 0), v100, z5, tool0;
	MoveL Offs(p0,602.5631999999999,93.1936, 0), v100, z5, tool0;
	MoveL Offs(p0,608.5046,101.74780000000001, 0), v100, z5, tool0;
	MoveL Offs(p0,613.6144,111.15520000000001, 0), v100, z5, tool0;
	MoveL Offs(p0,617.8578,121.38340000000001, 0), v100, z5, tool0;
	MoveL Offs(p0,621.2,132.4, 0), v100, z5, tool0;
	MoveL Offs(p0,622.5454000000001,138.83740000000003, 0), v100, z5, tool0;
	MoveL Offs(p0,623.4672000000003,145.93120000000005, 0), v100, z5, tool0;
	MoveL Offs(p0,623.9738,153.5338, 0), v100, z5, tool0;
	MoveL Offs(p0,624.0735999999999,161.4976, 0), v100, z5, tool0;
	MoveL Offs(p0,623.775,169.675, 0), v100, z5, tool0;
	MoveL Offs(p0,623.0864,177.9184, 0), v100, z5, tool0;
	MoveL Offs(p0,622.0162,186.08020000000002, 0), v100, z5, tool0;
	MoveL Offs(p0,620.5728000000001,194.01280000000003, 0), v100, z5, tool0;
	MoveL Offs(p0,618.7646,201.5686, 0), v100, z5, tool0;
	MoveL Offs(p0,616.6,208.6, 0), v100, z5, tool0;
	MoveL Offs(p0,612.6814,218.78920000000002, 0), v100, z5, tool0;
	MoveL Offs(p0,608.1232000000001,228.72160000000002, 0), v100, z5, tool0;
	MoveL Offs(p0,602.9218000000001,238.40439999999998, 0), v100, z5, tool0;
	MoveL Offs(p0,597.0736,247.84480000000002, 0), v100, z5, tool0;
	MoveL Offs(p0,590.575,257.05, 0), v100, z5, tool0;
	MoveL Offs(p0,583.4224,266.0272, 0), v100, z5, tool0;
	MoveL Offs(p0,575.6121999999999,274.78360000000004, 0), v100, z5, tool0;
	MoveL Offs(p0,567.1408,283.32640000000004, 0), v100, z5, tool0;
	MoveL Offs(p0,558.0046,291.6628, 0), v100, z5, tool0;
	MoveL Offs(p0,548.2,299.8, 0), v100, z5, tool0;
	MoveL Offs(p0,530.6,313.6, 0), v100, z5, tool0;
	MoveL Offs(p0,532.4,325.4, 0), v100, z5, tool0;
	MoveL Offs(p0,532.9526,329.4798, 0), v100, z5, tool0;
	MoveL Offs(p0,533.2928000000002,333.7744000000001, 0), v100, z5, tool0;
	MoveL Offs(p0,533.4242,338.24660000000006, 0), v100, z5, tool0;
	MoveL Offs(p0,533.3504,342.8592, 0), v100, z5, tool0;
	MoveL Offs(p0,533.075,347.575, 0), v100, z5, tool0;
	MoveL Offs(p0,532.6016,352.3568, 0), v100, z5, tool0;
	MoveL Offs(p0,531.9338,357.1674, 0), v100, z5, tool0;
	MoveL Offs(p0,531.0752,361.9696, 0), v100, z5, tool0;
	MoveL Offs(p0,530.0294000000001,366.7262, 0), v100, z5, tool0;
	MoveL Offs(p0,528.8,371.4, 0), v100, z5, tool0;
	MoveL Offs(p0,527.9542,374.43320000000006, 0), v100, z5, tool0;
	MoveL Offs(p0,527.3376000000001,377.0656000000001, 0), v100, z5, tool0;
	MoveL Offs(p0,526.9514,379.3164, 0), v100, z5, tool0;
	MoveL Offs(p0,526.7968000000001,381.2048000000001, 0), v100, z5, tool0;
	MoveL Offs(p0,526.875,382.75, 0), v100, z5, tool0;
	MoveL Offs(p0,527.1872,383.97119999999995, 0), v100, z5, tool0;
	MoveL Offs(p0,527.7346,384.8876, 0), v100, z5, tool0;
	MoveL Offs(p0,528.5184000000002,385.51840000000004, 0), v100, z5, tool0;
	MoveL Offs(p0,529.5398,385.88280000000003, 0), v100, z5, tool0;
	MoveL Offs(p0,530.8,386.0, 0), v100, z5, tool0;
	MoveL Offs(p0,534.4592000000001,382.3632000000001, 0), v100, z5, tool0;
	MoveL Offs(p0,537.4348,377.93780000000004, 0), v100, z5, tool0;
	MoveL Offs(p0,541.1136,371.88160000000005, 0), v100, z5, tool0;
	MoveL Offs(p0,545.45,364.275, 0), v100, z5, tool0;
	MoveL Offs(p0,550.3983999999999,355.19839999999994, 0), v100, z5, tool0;
	MoveL Offs(p0,555.9132,344.73220000000003, 0), v100, z5, tool0;
	MoveL Offs(p0,561.9488000000001,332.95680000000004, 0), v100, z5, tool0;
	MoveL Offs(p0,568.4595999999999,319.95259999999996, 0), v100, z5, tool0;
	MoveL Offs(p0,575.4,305.8, 0), v100, z5, tool0;
	MoveL Offs(p0,581.2984,293.84580000000005, 0), v100, z5, tool0;
	MoveL Offs(p0,586.3712000000003,283.8944000000001, 0), v100, z5, tool0;
	MoveL Offs(p0,590.7648,275.7525999999999, 0), v100, z5, tool0;
	MoveL Offs(p0,594.6256000000001,269.22720000000004, 0), v100, z5, tool0;
	MoveL Offs(p0,598.1,264.125, 0), v100, z5, tool0;
	MoveL Offs(p0,601.3344,260.2528, 0), v100, z5, tool0;
	MoveL Offs(p0,604.4752000000001,257.4174, 0), v100, z5, tool0;
	MoveL Offs(p0,607.6688,255.42560000000003, 0), v100, z5, tool0;
	MoveL Offs(p0,611.0616,254.0842, 0), v100, z5, tool0;
	MoveL Offs(p0,614.8,253.2, 0), v100, z5, tool0;
	MoveL Offs(p0,618.0974000000001,252.94320000000002, 0), v100, z5, tool0;
	MoveL Offs(p0,622.1232000000002,253.25760000000005, 0), v100, z5, tool0;
	MoveL Offs(p0,626.8978,254.1504, 0), v100, z5, tool0;
	MoveL Offs(p0,632.4416,255.6288, 0), v100, z5, tool0;
	MoveL Offs(p0,638.775,257.7, 0), v100, z5, tool0;
	MoveL Offs(p0,645.9183999999999,260.3712, 0), v100, z5, tool0;
	MoveL Offs(p0,653.8922,263.6496, 0), v100, z5, tool0;
	MoveL Offs(p0,662.7168,267.5424, 0), v100, z5, tool0;
	MoveL Offs(p0,672.4126,272.0568, 0), v100, z5, tool0;
	MoveL Offs(p0,683.0,277.2, 0), v100, z5, tool0;
	MoveL Offs(p0,694.0950000000001,282.79200000000003, 0), v100, z5, tool0;
	MoveL Offs(p0,703.6000000000003,287.7600000000001, 0), v100, z5, tool0;
	MoveL Offs(p0,711.665,292.212, 0), v100, z5, tool0;
	MoveL Offs(p0,718.4399999999999,296.256, 0), v100, z5, tool0;
	MoveL Offs(p0,724.075,300.0, 0), v100, z5, tool0;
	MoveL Offs(p0,728.72,303.55199999999996, 0), v100, z5, tool0;
	MoveL Offs(p0,732.525,307.02, 0), v100, z5, tool0;
	MoveL Offs(p0,735.6400000000001,310.512, 0), v100, z5, tool0;
	MoveL Offs(p0,738.2149999999999,314.136, 0), v100, z5, tool0;
	MoveL Offs(p0,740.4,318.0, 0), v100, z5, tool0;
	MoveL Offs(p0,743.1044,323.64080000000007, 0), v100, z5, tool0;
	MoveL Offs(p0,744.8752000000002,328.9744000000001, 0), v100, z5, tool0;
	MoveL Offs(p0,745.5588,334.43760000000003, 0), v100, z5, tool0;
	MoveL Offs(p0,745.0016,340.4672000000001, 0), v100, z5, tool0;
	MoveL Offs(p0,743.05,347.5, 0), v100, z5, tool0;
	MoveL Offs(p0,739.5504000000001,355.97279999999995, 0), v100, z5, tool0;
	MoveL Offs(p0,734.3492,366.3224, 0), v100, z5, tool0;
	MoveL Offs(p0,727.2928,378.98560000000003, 0), v100, z5, tool0;
	MoveL Offs(p0,718.2275999999999,394.3992, 0), v100, z5, tool0;
	MoveL Offs(p0,707.0,413.0, 0), v100, z5, tool0;
	MoveL Offs(p0,702.8460000000001,419.9014000000001, 0), v100, z5, tool0;
	MoveL Offs(p0,698.8240000000002,426.6192000000002, 0), v100, z5, tool0;
	MoveL Offs(p0,694.9939999999999,433.05379999999997, 0), v100, z5, tool0;
	MoveL Offs(p0,691.416,439.1056, 0), v100, z5, tool0;
	MoveL Offs(p0,688.15,444.675, 0), v100, z5, tool0;
	MoveL Offs(p0,685.2560000000001,449.6624, 0), v100, z5, tool0;
	MoveL Offs(p0,682.7940000000001,453.96819999999997, 0), v100, z5, tool0;
	MoveL Offs(p0,680.824,457.4928, 0), v100, z5, tool0;
	MoveL Offs(p0,679.4060000000001,460.1366, 0), v100, z5, tool0;
	MoveL Offs(p0,678.6,461.8, 0), v100, z5, tool0;
	MoveL Offs(p0,677.2704000000001,465.0896000000001, 0), v100, z5, tool0;
	MoveL Offs(p0,676.8846000000001,466.3143999999999, 0), v100, z5, tool0;
	MoveL Offs(p0,676.6992,467.33280000000013, 0), v100, z5, tool0;
	MoveL Offs(p0,676.725,468.2, 0), v100, z5, tool0;
	MoveL Offs(p0,676.9728,468.97119999999995, 0), v100, z5, tool0;
	MoveL Offs(p0,677.4534,469.7016, 0), v100, z5, tool0;
	MoveL Offs(p0,678.1776000000001,470.4464, 0), v100, z5, tool0;
	MoveL Offs(p0,679.1562000000001,471.2608, 0), v100, z5, tool0;
	MoveL Offs(p0,680.4,472.2, 0), v100, z5, tool0;
	MoveL Offs(p0,684.1148000000001,474.61260000000004, 0), v100, z5, tool0;
	MoveL Offs(p0,688.1344000000001,476.4528000000002, 0), v100, z5, tool0;
	MoveL Offs(p0,692.3916,477.72419999999994, 0), v100, z5, tool0;
	MoveL Offs(p0,696.8192000000001,478.4304, 0), v100, z5, tool0;
	MoveL Offs(p0,701.35,478.575, 0), v100, z5, tool0;
	MoveL Offs(p0,705.9168,478.1616, 0), v100, z5, tool0;
	MoveL Offs(p0,710.4523999999999,477.1938, 0), v100, z5, tool0;
	MoveL Offs(p0,714.8896000000001,475.6752, 0), v100, z5, tool0;
	MoveL Offs(p0,719.1612,473.6094000000001, 0), v100, z5, tool0;
	MoveL Offs(p0,723.2,471.0, 0), v100, z5, tool0;
	MoveL Offs(p0,725.4206000000001,468.98160000000007, 0), v100, z5, tool0;
	MoveL Offs(p0,727.7408000000003,466.32480000000004, 0), v100, z5, tool0;
	MoveL Offs(p0,730.1281999999999,463.08719999999994, 0), v100, z5, tool0;
	MoveL Offs(p0,732.5504000000001,459.32640000000004, 0), v100, z5, tool0;
	MoveL Offs(p0,734.975,455.1, 0), v100, z5, tool0;
	MoveL Offs(p0,737.3696,450.4656, 0), v100, z5, tool0;
	MoveL Offs(p0,739.7018,445.4808, 0), v100, z5, tool0;
	MoveL Offs(p0,741.9392,440.20320000000004, 0), v100, z5, tool0;
	MoveL Offs(p0,744.0494000000001,434.69040000000007, 0), v100, z5, tool0;
	MoveL Offs(p0,746.0,429.0, 0), v100, z5, tool0;
	MoveL Offs(p0,751.7486000000001,412.721, 0), v100, z5, tool0;
	MoveL Offs(p0,758.4128000000003,397.62400000000014, 0), v100, z5, tool0;
	MoveL Offs(p0,765.9602,383.739, 0), v100, z5, tool0;
	MoveL Offs(p0,774.3584,371.09600000000006, 0), v100, z5, tool0;
	MoveL Offs(p0,783.575,359.725, 0), v100, z5, tool0;
	MoveL Offs(p0,793.5776,349.656, 0), v100, z5, tool0;
	MoveL Offs(p0,804.3338,340.919, 0), v100, z5, tool0;
	MoveL Offs(p0,815.8112,333.54400000000004, 0), v100, z5, tool0;
	MoveL Offs(p0,827.9774000000001,327.561, 0), v100, z5, tool0;
	MoveL Offs(p0,840.8,323.0, 0), v100, z5, tool0;
	MoveL Offs(p0,846.3076000000001,321.696, 0), v100, z5, tool0;
	MoveL Offs(p0,852.6048000000001,320.7760000000001, 0), v100, z5, tool0;
	MoveL Offs(p0,859.4732,320.22799999999995, 0), v100, z5, tool0;
	MoveL Offs(p0,866.6944,320.04, 0), v100, z5, tool0;
	MoveL Offs(p0,874.05,320.2, 0), v100, z5, tool0;
	MoveL Offs(p0,881.3216,320.696, 0), v100, z5, tool0;
	MoveL Offs(p0,888.2908,321.51599999999996, 0), v100, z5, tool0;
	MoveL Offs(p0,894.7392,322.648, 0), v100, z5, tool0;
	MoveL Offs(p0,900.4484,324.08000000000004, 0), v100, z5, tool0;
	MoveL Offs(p0,905.2,325.8, 0), v100, z5, tool0;
	MoveL Offs(p0,908.8114000000002,327.56360000000006, 0), v100, z5, tool0;
	MoveL Offs(p0,912.4192000000003,329.7088000000001, 0), v100, z5, tool0;
	MoveL Offs(p0,915.9838,332.19719999999995, 0), v100, z5, tool0;
	MoveL Offs(p0,919.4656000000001,334.9904, 0), v100, z5, tool0;
	MoveL Offs(p0,922.825,338.05, 0), v100, z5, tool0;
	MoveL Offs(p0,926.0224000000001,341.3376, 0), v100, z5, tool0;
	MoveL Offs(p0,929.0182000000001,344.8148, 0), v100, z5, tool0;
	MoveL Offs(p0,931.7728000000001,348.44320000000005, 0), v100, z5, tool0;
	MoveL Offs(p0,934.2466000000001,352.1844, 0), v100, z5, tool0;
	MoveL Offs(p0,936.4,356.0, 0), v100, z5, tool0;
	MoveL Offs(p0,938.2300000000001,360.2532, 0), v100, z5, tool0;
	MoveL Offs(p0,939.6400000000003,365.01760000000013, 0), v100, z5, tool0;
	MoveL Offs(p0,940.6299999999999,370.18039999999996, 0), v100, z5, tool0;
	MoveL Offs(p0,941.2,375.6288, 0), v100, z5, tool0;
	MoveL Offs(p0,941.35,381.25, 0), v100, z5, tool0;
	MoveL Offs(p0,941.0799999999999,386.9312, 0), v100, z5, tool0;
	MoveL Offs(p0,940.39,392.55959999999993, 0), v100, z5, tool0;
	MoveL Offs(p0,939.28,398.0224, 0), v100, z5, tool0;
	MoveL Offs(p0,937.75,403.20680000000004, 0), v100, z5, tool0;
	MoveL Offs(p0,935.8,408.0, 0), v100, z5, tool0;
	MoveL Offs(p0,932.0128000000001,415.0892, 0), v100, z5, tool0;
	MoveL Offs(p0,927.4144000000002,421.9216000000001, 0), v100, z5, tool0;
	MoveL Offs(p0,922.0695999999998,428.4444, 0), v100, z5, tool0;
	MoveL Offs(p0,916.0432000000001,434.60479999999995, 0), v100, z5, tool0;
	MoveL Offs(p0,909.4,440.35, 0), v100, z5, tool0;
	MoveL Offs(p0,902.2048000000001,445.6272, 0), v100, z5, tool0;
	MoveL Offs(p0,894.5223999999998,450.3836, 0), v100, z5, tool0;
	MoveL Offs(p0,886.4176,454.56640000000004, 0), v100, z5, tool0;
	MoveL Offs(p0,877.9552,458.1228, 0), v100, z5, tool0;
	MoveL Offs(p0,869.2,461.0, 0), v100, z5, tool0;
	MoveL Offs(p0,861.7162000000001,462.7302000000001, 0), v100, z5, tool0;
	MoveL Offs(p0,853.7536000000002,463.7536000000002, 0), v100, z5, tool0;
	MoveL Offs(p0,845.6254000000001,464.11940000000004, 0), v100, z5, tool0;
	MoveL Offs(p0,837.6448000000003,463.8768, 0), v100, z5, tool0;
	MoveL Offs(p0,830.125,463.075, 0), v100, z5, tool0;
	MoveL Offs(p0,823.3792000000001,461.7632, 0), v100, z5, tool0;
	MoveL Offs(p0,817.7206,459.9906, 0), v100, z5, tool0;
	MoveL Offs(p0,813.4624000000001,457.80640000000005, 0), v100, z5, tool0;
	MoveL Offs(p0,810.9177999999999,455.2598, 0), v100, z5, tool0;
	MoveL Offs(p0,810.4,452.4, 0), v100, z5, tool0;
	MoveL Offs(p0,812.6481999999999,450.0186, 0), v100, z5, tool0;
	MoveL Offs(p0,814.1824,449.6032, 0), v100, z5, tool0;
	MoveL Offs(p0,816.175,449.375, 0), v100, z5, tool0;
	MoveL Offs(p0,818.6656,449.3328, 0), v100, z5, tool0;
	MoveL Offs(p0,821.6938,449.4754, 0), v100, z5, tool0;
	MoveL Offs(p0,825.2992,449.80159999999995, 0), v100, z5, tool0;
	MoveL Offs(p0,829.5214,450.31020000000007, 0), v100, z5, tool0;
	MoveL Offs(p0,834.4,451.0, 0), v100, z5, tool0;
	MoveL Offs(p0,839.8226000000001,451.427, 0), v100, z5, tool0;
	MoveL Offs(p0,845.6928000000004,451.1760000000001, 0), v100, z5, tool0;
	MoveL Offs(p0,851.8942,450.28900000000004, 0), v100, z5, tool0;
	MoveL Offs(p0,858.3104000000001,448.808, 0), v100, z5, tool0;
	MoveL Offs(p0,864.825,446.775, 0), v100, z5, tool0;
	MoveL Offs(p0,871.3216,444.23199999999997, 0), v100, z5, tool0;
	MoveL Offs(p0,877.6838,441.221, 0), v100, z5, tool0;
	MoveL Offs(p0,883.7952000000001,437.784, 0), v100, z5, tool0;
	MoveL Offs(p0,889.5394,433.963, 0), v100, z5, tool0;
	MoveL Offs(p0,894.8,429.8, 0), v100, z5, tool0;
	MoveL Offs(p0,897.9932000000001,426.783, 0), v100, z5, tool0;
	MoveL Offs(p0,901.0736000000003,423.52000000000015, 0), v100, z5, tool0;
	MoveL Offs(p0,904.0124,420.053, 0), v100, z5, tool0;
	MoveL Offs(p0,906.7808000000001,416.4240000000001, 0), v100, z5, tool0;
	MoveL Offs(p0,909.35,412.675, 0), v100, z5, tool0;
	MoveL Offs(p0,911.6912,408.848, 0), v100, z5, tool0;
	MoveL Offs(p0,913.7755999999999,404.985, 0), v100, z5, tool0;
	MoveL Offs(p0,915.5744000000001,401.12800000000004, 0), v100, z5, tool0;
	MoveL Offs(p0,917.0588,397.3190000000001, 0), v100, z5, tool0;
	MoveL Offs(p0,918.2,393.6, 0), v100, z5, tool0;
	MoveL Offs(p0,919.3876000000002,382.7688000000001, 0), v100, z5, tool0;
	MoveL Offs(p0,917.2368000000002,372.8544000000001, 0), v100, z5, tool0;
	MoveL Offs(p0,912.1771999999999,364.0656, 0), v100, z5, tool0;
	MoveL Offs(p0,904.6384,356.6112, 0), v100, z5, tool0;
	MoveL Offs(p0,895.05,350.7, 0), v100, z5, tool0;
	MoveL Offs(p0,883.8416,346.54079999999993, 0), v100, z5, tool0;
	MoveL Offs(p0,871.4428,344.3424, 0), v100, z5, tool0;
	MoveL Offs(p0,858.2832000000001,344.31360000000006, 0), v100, z5, tool0;
	MoveL Offs(p0,844.7924,346.6632, 0), v100, z5, tool0;
	MoveL Offs(p0,831.4,351.6, 0), v100, z5, tool0;
	MoveL Offs(p0,823.3034000000001,355.87840000000006, 0), v100, z5, tool0;
	MoveL Offs(p0,815.7792000000003,360.96320000000014, 0), v100, z5, tool0;
	MoveL Offs(p0,808.7758,366.9288, 0), v100, z5, tool0;
	MoveL Offs(p0,802.2416000000001,373.8496, 0), v100, z5, tool0;
	MoveL Offs(p0,796.125,381.8, 0), v100, z5, tool0;
	MoveL Offs(p0,790.3743999999999,390.85440000000006, 0), v100, z5, tool0;
	MoveL Offs(p0,784.9381999999999,401.08720000000005, 0), v100, z5, tool0;
	MoveL Offs(p0,779.7648000000002,412.57280000000003, 0), v100, z5, tool0;
	MoveL Offs(p0,774.8026000000001,425.38559999999995, 0), v100, z5, tool0;
	MoveL Offs(p0,770.0,439.6, 0), v100, z5, tool0;
	MoveL Offs(p0,768.3264000000001,444.6752, 0), v100, z5, tool0;
	MoveL Offs(p0,766.6672000000002,449.45760000000007, 0), v100, z5, tool0;
	MoveL Offs(p0,765.0247999999999,453.9423999999999, 0), v100, z5, tool0;
	MoveL Offs(p0,763.4016,458.12480000000005, 0), v100, z5, tool0;
	MoveL Offs(p0,761.8,462.0, 0), v100, z5, tool0;
	MoveL Offs(p0,760.2224,465.56319999999994, 0), v100, z5, tool0;
	MoveL Offs(p0,758.6712,468.80959999999993, 0), v100, z5, tool0;
	MoveL Offs(p0,757.1488,471.7344000000001, 0), v100, z5, tool0;
	MoveL Offs(p0,755.6576,474.33279999999996, 0), v100, z5, tool0;
	MoveL Offs(p0,754.2,476.6, 0), v100, z5, tool0;
	MoveL Offs(p0,751.5624000000001,480.0924000000001, 0), v100, z5, tool0;
	MoveL Offs(p0,748.6032000000002,483.46720000000016, 0), v100, z5, tool0;
	MoveL Offs(p0,745.3728,486.69079999999997, 0), v100, z5, tool0;
	MoveL Offs(p0,741.9215999999999,489.7296, 0), v100, z5, tool0;
	MoveL Offs(p0,738.3,492.55, 0), v100, z5, tool0;
	MoveL Offs(p0,734.5584,495.1184, 0), v100, z5, tool0;
	MoveL Offs(p0,730.7472,497.40119999999996, 0), v100, z5, tool0;
	MoveL Offs(p0,726.9168000000001,499.3648000000001, 0), v100, z5, tool0;
	MoveL Offs(p0,723.1176,500.97560000000004, 0), v100, z5, tool0;
	MoveL Offs(p0,719.4,502.2, 0), v100, z5, tool0;
	MoveL Offs(p0,716.4294000000001,502.825, 0), v100, z5, tool0;
	MoveL Offs(p0,712.7952000000001,503.26400000000024, 0), v100, z5, tool0;
	MoveL Offs(p0,708.6738,503.52299999999997, 0), v100, z5, tool0;
	MoveL Offs(p0,704.2416000000001,503.608, 0), v100, z5, tool0;
	MoveL Offs(p0,699.675,503.525, 0), v100, z5, tool0;
	MoveL Offs(p0,695.1504,503.28000000000003, 0), v100, z5, tool0;
	MoveL Offs(p0,690.8441999999999,502.879, 0), v100, z5, tool0;
	MoveL Offs(p0,686.9328,502.3280000000001, 0), v100, z5, tool0;
	MoveL Offs(p0,683.5926000000001,501.633, 0), v100, z5, tool0;
	MoveL Offs(p0,681.0,500.8, 0), v100, z5, tool0;
	MoveL Offs(p0,678.6995999999999,500.0044, 0), v100, z5, tool0;
	MoveL Offs(p0,678.3312000000001,499.9648, 0), v100, z5, tool0;
	MoveL Offs(p0,678.15,500.05, 0), v100, z5, tool0;
	MoveL Offs(p0,678.1487999999999,500.26720000000006, 0), v100, z5, tool0;
	MoveL Offs(p0,678.3204,500.6236, 0), v100, z5, tool0;
	MoveL Offs(p0,678.6576000000001,501.1264000000001, 0), v100, z5, tool0;
	MoveL Offs(p0,683.1974,505.36220000000014, 0), v100, z5, tool0;
	MoveL Offs(p0,688.5952000000002,507.9696000000002, 0), v100, z5, tool0;
	MoveL Offs(p0,695.6418,510.3634, 0), v100, z5, tool0;
	MoveL Offs(p0,703.9856,512.4848000000001, 0), v100, z5, tool0;
	MoveL Offs(p0,713.275,514.275, 0), v100, z5, tool0;
	MoveL Offs(p0,723.1584,515.6752, 0), v100, z5, tool0;
	MoveL Offs(p0,733.2841999999999,516.6266, 0), v100, z5, tool0;
	MoveL Offs(p0,743.3008000000001,517.0704000000001, 0), v100, z5, tool0;
	MoveL Offs(p0,752.8566,516.9478, 0), v100, z5, tool0;
	MoveL Offs(p0,761.6,516.2, 0), v100, z5, tool0;
	MoveL Offs(p0,768.3124,515.3936000000001, 0), v100, z5, tool0;
	MoveL Offs(p0,773.8032000000002,514.7888000000002, 0), v100, z5, tool0;
	MoveL Offs(p0,778.2428,514.4072, 0), v100, z5, tool0;
	MoveL Offs(p0,781.8016000000001,514.2704000000001, 0), v100, z5, tool0;
	MoveL Offs(p0,784.65,514.4, 0), v100, z5, tool0;
	MoveL Offs(p0,786.9584,514.8176, 0), v100, z5, tool0;
	MoveL Offs(p0,788.8972,515.5448, 0), v100, z5, tool0;
	MoveL Offs(p0,790.6368,516.6032000000001, 0), v100, z5, tool0;
	MoveL Offs(p0,792.3476,518.0144, 0), v100, z5, tool0;
	MoveL Offs(p0,794.2,519.8, 0), v100, z5, tool0;
	MoveL Offs(p0,796.6536000000002,522.5464000000001, 0), v100, z5, tool0;
	MoveL Offs(p0,798.4928000000002,525.2832000000001, 0), v100, z5, tool0;
	MoveL Offs(p0,799.7152,528.0368, 0), v100, z5, tool0;
	MoveL Offs(p0,800.3184,530.8336, 0), v100, z5, tool0;
	MoveL Offs(p0,800.3,533.7, 0), v100, z5, tool0;
	MoveL Offs(p0,799.6575999999999,536.6623999999999, 0), v100, z5, tool0;
	MoveL Offs(p0,798.3888000000001,539.7472, 0), v100, z5, tool0;
	MoveL Offs(p0,796.4912,542.9808, 0), v100, z5, tool0;
	MoveL Offs(p0,793.9624,546.3896000000001, 0), v100, z5, tool0;
	MoveL Offs(p0,790.8,550.0, 0), v100, z5, tool0;
	MoveL Offs(p0,787.4084000000001,553.8624000000001, 0), v100, z5, tool0;
	MoveL Offs(p0,784.6672000000002,557.5712000000001, 0), v100, z5, tool0;
	MoveL Offs(p0,782.5668000000001,561.1888, 0), v100, z5, tool0;
	MoveL Offs(p0,781.0976000000002,564.7776, 0), v100, z5, tool0;
	MoveL Offs(p0,780.25,568.4, 0), v100, z5, tool0;
	MoveL Offs(p0,780.0144,572.1184000000001, 0), v100, z5, tool0;
	MoveL Offs(p0,780.3812,575.9952000000001, 0), v100, z5, tool0;
	MoveL Offs(p0,781.3408000000002,580.0928000000001, 0), v100, z5, tool0;
	MoveL Offs(p0,782.8836,584.4736, 0), v100, z5, tool0;
	MoveL Offs(p0,785.0,589.2, 0), v100, z5, tool0;
	MoveL Offs(p0,786.9722,592.8416, 0), v100, z5, tool0;
	MoveL Offs(p0,789.1136000000002,596.1328000000002, 0), v100, z5, tool0;
	MoveL Offs(p0,791.5214000000001,599.1432, 0), v100, z5, tool0;
	MoveL Offs(p0,794.2928000000002,601.9424, 0), v100, z5, tool0;
	MoveL Offs(p0,797.525,604.6, 0), v100, z5, tool0;
	MoveL Offs(p0,801.3152,607.1856, 0), v100, z5, tool0;
	MoveL Offs(p0,805.7606,609.7688, 0), v100, z5, tool0;
	MoveL Offs(p0,810.9584000000001,612.4192, 0), v100, z5, tool0;
	MoveL Offs(p0,817.0058000000001,615.2064, 0), v100, z5, tool0;
	MoveL Offs(p0,824.0,618.2, 0), v100, z5, tool0;
	MoveL Offs(p0,826.6448,619.3184000000001, 0), v100, z5, tool0;
	MoveL Offs(p0,829.2704000000001,620.4992000000002, 0), v100, z5, tool0;
	MoveL Offs(p0,831.8335999999999,621.7207999999999, 0), v100, z5, tool0;
	MoveL Offs(p0,834.2912,622.9616000000001, 0), v100, z5, tool0;
	MoveL Offs(p0,836.6,624.2, 0), v100, z5, tool0;
	MoveL Offs(p0,838.7167999999999,625.4143999999999, 0), v100, z5, tool0;
	MoveL Offs(p0,840.5984000000001,626.5832, 0), v100, z5, tool0;
	MoveL Offs(p0,842.2016000000001,627.6848000000001, 0), v100, z5, tool0;
	MoveL Offs(p0,843.4832,628.6976000000001, 0), v100, z5, tool0;
	MoveL Offs(p0,844.4,629.6, 0), v100, z5, tool0;
	MoveL Offs(p0,846.2602,631.8902, 0), v100, z5, tool0;
	MoveL Offs(p0,847.6416000000003,634.4336000000001, 0), v100, z5, tool0;
	MoveL Offs(p0,848.5454,637.2194, 0), v100, z5, tool0;
	MoveL Offs(p0,848.9728000000001,640.2368, 0), v100, z5, tool0;
	MoveL Offs(p0,848.925,643.475, 0), v100, z5, tool0;
	MoveL Offs(p0,848.4032000000001,646.9232, 0), v100, z5, tool0;
	MoveL Offs(p0,847.4086,650.5706, 0), v100, z5, tool0;
	MoveL Offs(p0,845.9424000000001,654.4064000000001, 0), v100, z5, tool0;
	MoveL Offs(p0,844.0058000000001,658.4198, 0), v100, z5, tool0;
	MoveL Offs(p0,841.6,662.6, 0), v100, z5, tool0;
	MoveL Offs(p0,838.9212000000001,667.1424000000001, 0), v100, z5, tool0;
	MoveL Offs(p0,836.6336000000003,671.5792000000001, 0), v100, z5, tool0;
	MoveL Offs(p0,834.7203999999999,675.9848, 0), v100, z5, tool0;
	MoveL Offs(p0,833.1648000000001,680.4336000000001, 0), v100, z5, tool0;
	MoveL Offs(p0,831.95,685.0, 0), v100, z5, tool0;
	MoveL Offs(p0,831.0592,689.7583999999999, 0), v100, z5, tool0;
	MoveL Offs(p0,830.4756,694.7832, 0), v100, z5, tool0;
	MoveL Offs(p0,830.1824,700.1488, 0), v100, z5, tool0;
	MoveL Offs(p0,830.1628000000001,705.9296, 0), v100, z5, tool0;
	MoveL Offs(p0,830.4,712.2, 0), v100, z5, tool0;
	MoveL Offs(p0,831.0154,719.1544000000001, 0), v100, z5, tool0;
	MoveL Offs(p0,832.0112000000003,725.7152000000002, 0), v100, z5, tool0;
	MoveL Offs(p0,833.3718000000001,731.8488, 0), v100, z5, tool0;
	MoveL Offs(p0,835.0816000000001,737.5216, 0), v100, z5, tool0;
	MoveL Offs(p0,837.125,742.7, 0), v100, z5, tool0;
	MoveL Offs(p0,839.4864,747.3503999999999, 0), v100, z5, tool0;
	MoveL Offs(p0,842.1502,751.4392, 0), v100, z5, tool0;
	MoveL Offs(p0,845.1008000000002,754.9328, 0), v100, z5, tool0;
	MoveL Offs(p0,848.3226000000001,757.7976000000001, 0), v100, z5, tool0;
	MoveL Offs(p0,851.8,760.0, 0), v100, z5, tool0;
	MoveL Offs(p0,854.3676000000002,761.4332, 0), v100, z5, tool0;
	MoveL Offs(p0,856.5488000000001,762.9696000000001, 0), v100, z5, tool0;
	MoveL Offs(p0,858.3412000000001,764.6043999999999, 0), v100, z5, tool0;
	MoveL Offs(p0,859.7424000000001,766.3328000000001, 0), v100, z5, tool0;
	MoveL Offs(p0,860.75,768.15, 0), v100, z5, tool0;
	MoveL Offs(p0,861.3616,770.0512, 0), v100, z5, tool0;
	MoveL Offs(p0,861.5748,772.0316, 0), v100, z5, tool0;
	MoveL Offs(p0,861.3872000000001,774.0864, 0), v100, z5, tool0;
	MoveL Offs(p0,860.7964,776.2108000000001, 0), v100, z5, tool0;
	MoveL Offs(p0,859.8,778.4, 0), v100, z5, tool0;
	MoveL Offs(p0,858.0160000000003,781.4944000000003, 0), v100, z5, tool0;
	MoveL Offs(p0,857.1,782.6876, 0), v100, z5, tool0;
	MoveL Offs(p0,856.1360000000001,783.6672000000001, 0), v100, z5, tool0;
	MoveL Offs(p0,855.1,784.45, 0), v100, z5, tool0;
	MoveL Offs(p0,853.9679999999998,785.0527999999999, 0), v100, z5, tool0;
	MoveL Offs(p0,852.716,785.4924, 0), v100, z5, tool0;
	MoveL Offs(p0,851.32,785.7856000000002, 0), v100, z5, tool0;
	MoveL Offs(p0,849.7560000000001,785.9492, 0), v100, z5, tool0;
	MoveL Offs(p0,848.0,786.0, 0), v100, z5, tool0;
	MoveL Offs(p0,843.7982000000002,784.9684000000001, 0), v100, z5, tool0;
	MoveL Offs(p0,837.2576000000001,781.9952000000002, 0), v100, z5, tool0;
	MoveL Offs(p0,828.6553999999999,777.2628, 0), v100, z5, tool0;
	MoveL Offs(p0,818.2688,770.9536, 0), v100, z5, tool0;
	MoveL Offs(p0,806.375,763.25, 0), v100, z5, tool0;
	MoveL Offs(p0,793.2511999999999,754.3344, 0), v100, z5, tool0;
	MoveL Offs(p0,779.1746,744.3892, 0), v100, z5, tool0;
	MoveL Offs(p0,764.4224,733.5968, 0), v100, z5, tool0;
	MoveL Offs(p0,749.2718,722.1396000000001, 0), v100, z5, tool0;
	MoveL Offs(p0,734.0,710.2, 0), v100, z5, tool0;
	MoveL Offs(p0,709.0,690.4, 0), v100, z5, tool0;
	MoveL Offs(p0,707.4,696.4, 0), v100, z5, tool0;
	MoveL Offs(p0,706.0678,700.6246000000001, 0), v100, z5, tool0;
	MoveL Offs(p0,704.4704000000002,704.1808000000002, 0), v100, z5, tool0;
	MoveL Offs(p0,702.6066000000001,707.0722, 0), v100, z5, tool0;
	MoveL Offs(p0,700.4752000000001,709.3024000000001, 0), v100, z5, tool0;
	MoveL Offs(p0,698.075,710.875, 0), v100, z5, tool0;
	MoveL Offs(p0,695.4048,711.7936, 0), v100, z5, tool0;
	MoveL Offs(p0,692.4634,712.0618000000001, 0), v100, z5, tool0;
	MoveL Offs(p0,689.2496000000001,711.6832, 0), v100, z5, tool0;
	MoveL Offs(p0,685.7622,710.6614, 0), v100, z5, tool0;
	MoveL Offs(p0,682.0,709.0, 0), v100, z5, tool0;
	MoveL Offs(p0,679.6096000000002,707.8240000000002, 0), v100, z5, tool0;
	MoveL Offs(p0,678.6754,707.434, 0), v100, z5, tool0;
	MoveL Offs(p0,677.9008000000001,707.176, 0), v100, z5, tool0;
	MoveL Offs(p0,677.275,707.05, 0), v100, z5, tool0;
	MoveL Offs(p0,676.7872,707.0559999999999, 0), v100, z5, tool0;
	MoveL Offs(p0,676.4266,707.1940000000001, 0), v100, z5, tool0;
	MoveL Offs(p0,676.1824,707.464, 0), v100, z5, tool0;
	MoveL Offs(p0,676.0438,707.866, 0), v100, z5, tool0;
	MoveL Offs(p0,676.0,708.4, 0), v100, z5, tool0;
	MoveL Offs(p0,675.8740000000001,710.4966000000002, 0), v100, z5, tool0;
	MoveL Offs(p0,675.5200000000001,712.7648000000002, 0), v100, z5, tool0;
	MoveL Offs(p0,674.9739999999999,715.1122, 0), v100, z5, tool0;
	MoveL Offs(p0,674.272,717.4464, 0), v100, z5, tool0;
	MoveL Offs(p0,673.45,719.675, 0), v100, z5, tool0;
	MoveL Offs(p0,672.5439999999999,721.7056, 0), v100, z5, tool0;
	MoveL Offs(p0,671.5899999999999,723.4458000000001, 0), v100, z5, tool0;
	MoveL Offs(p0,670.624,724.8032000000001, 0), v100, z5, tool0;
	MoveL Offs(p0,669.682,725.6854000000001, 0), v100, z5, tool0;
	MoveL Offs(p0,668.8,726.0, 0), v100, z5, tool0;
	MoveL Offs(p0,666.5040000000001,725.4784000000002, 0), v100, z5, tool0;
	MoveL Offs(p0,664.4440000000001,724.8605999999999, 0), v100, z5, tool0;
	MoveL Offs(p0,661.856,724.0351999999999, 0), v100, z5, tool0;
	MoveL Offs(p0,658.8,723.025, 0), v100, z5, tool0;
	MoveL Offs(p0,655.336,721.8528, 0), v100, z5, tool0;
	MoveL Offs(p0,651.524,720.5414000000001, 0), v100, z5, tool0;
	MoveL Offs(p0,647.4240000000001,719.1136, 0), v100, z5, tool0;
	MoveL Offs(p0,643.096,717.5922, 0), v100, z5, tool0;
	MoveL Offs(p0,638.6,716.0, 0), v100, z5, tool0;
	MoveL Offs(p0,634.1876,714.365, 0), v100, z5, tool0;
	MoveL Offs(p0,629.9888000000002,712.8320000000001, 0), v100, z5, tool0;
	MoveL Offs(p0,626.0612,711.419, 0), v100, z5, tool0;
	MoveL Offs(p0,622.4624000000001,710.1440000000001, 0), v100, z5, tool0;
	MoveL Offs(p0,619.25,709.025, 0), v100, z5, tool0;
	MoveL Offs(p0,616.4816000000001,708.0799999999999, 0), v100, z5, tool0;
	MoveL Offs(p0,614.2148,707.327, 0), v100, z5, tool0;
	MoveL Offs(p0,612.5072,706.784, 0), v100, z5, tool0;
	MoveL Offs(p0,611.4164000000001,706.469, 0), v100, z5, tool0;
	MoveL Offs(p0,611.0,706.4, 0), v100, z5, tool0;
	MoveL Offs(p0,612.6722000000001,710.189, 0), v100, z5, tool0;
	MoveL Offs(p0,613.9664,712.8, 0), v100, z5, tool0;
	MoveL Offs(p0,615.575,715.975, 0), v100, z5, tool0;
	MoveL Offs(p0,617.4655999999999,719.6479999999999, 0), v100, z5, tool0;
	MoveL Offs(p0,619.6058,723.753, 0), v100, z5, tool0;
	MoveL Offs(p0,621.9631999999999,728.2239999999999, 0), v100, z5, tool0;
	MoveL Offs(p0,624.5054,732.995, 0), v100, z5, tool0;
	MoveL Offs(p0,627.2,738.0, 0), v100, z5, tool0;
	MoveL Offs(p0,630.6296,744.4214, 0), v100, z5, tool0;
	MoveL Offs(p0,633.6128000000002,750.1552000000001, 0), v100, z5, tool0;
	MoveL Offs(p0,636.1712,755.2457999999999, 0), v100, z5, tool0;
	MoveL Offs(p0,638.3264,759.7376000000002, 0), v100, z5, tool0;
	MoveL Offs(p0,640.1,763.675, 0), v100, z5, tool0;
	MoveL Offs(p0,641.5136,767.1024, 0), v100, z5, tool0;
	MoveL Offs(p0,642.5887999999999,770.0642, 0), v100, z5, tool0;
	MoveL Offs(p0,643.3471999999999,772.6048000000001, 0), v100, z5, tool0;
	MoveL Offs(p0,643.8104,774.7686, 0), v100, z5, tool0;
	MoveL Offs(p0,644.0,776.6, 0), v100, z5, tool0;
	MoveL Offs(p0,643.7152000000001,780.0856, 0), v100, z5, tool0;
	MoveL Offs(p0,642.8976000000002,783.1968000000002, 0), v100, z5, tool0;
	MoveL Offs(p0,641.6024,785.8952, 0), v100, z5, tool0;
	MoveL Offs(p0,639.8848,788.1424000000001, 0), v100, z5, tool0;
	MoveL Offs(p0,637.8,789.9, 0), v100, z5, tool0;
	MoveL Offs(p0,635.4032,791.1296, 0), v100, z5, tool0;
	MoveL Offs(p0,632.7495999999999,791.7927999999999, 0), v100, z5, tool0;
	MoveL Offs(p0,629.8944,791.8512000000001, 0), v100, z5, tool0;
	MoveL Offs(p0,626.8928,791.2664, 0), v100, z5, tool0;
